// 2. Fallback handling
IF VO_Error THEN
    IF VI_Fallback_Mode = 1 THEN
        VO_Value := VI_Default_Value;
    END_IF;
    // If VI_Fallback_Mode = 0, VO_Value retains its last good value (L_Filtered)
    RETURN;
END_IF;

// 3. Calibration
L_Scaled := (L_Scaled * VI_Multiplier) + VI_Offset;

// 4. Moving Average Filter (ТЗ 1.2)
IF L_First_Scan THEN
    L_Filtered := L_Scaled;
    L_First_Scan := FALSE;
    L_Last_Time := VI_System_Time_MS;
    
    // Инициализация массива истории
    FOR L_i := 0 TO 9 DO
        L_History[L_i] := L_Scaled;
    END_FOR;
    L_History_Sum := L_Scaled * 10.0;
    L_History_Count := 10;
    L_History_Idx := 0;
END_IF;

L_DT := (SEL(VI_System_Time_MS >= L_Last_Time, VI_System_Time_MS - L_Last_Time, (4294967295 - L_Last_Time) + VI_System_Time_MS + 1));
IF VI_Filter_Time_MS = 0 THEN
    L_Filtered := L_Scaled;
    L_Last_Time := VI_System_Time_MS;
ELSIF L_DT >= (VI_Filter_Time_MS / 10) THEN // Обновляем 10 раз за время фильтрации
    // Вычитаем старое значение
    L_History_Sum := L_History_Sum - L_History[L_History_Idx];
    
    // Добавляем новое значение
    L_History[L_History_Idx] := L_Scaled;
    L_History_Sum := L_History_Sum + L_Scaled;
    
    // Сдвигаем индекс
    L_History_Idx := (L_History_Idx + 1) MOD 10;
    
    // Вычисляем среднее
    L_Filtered := L_History_Sum / 10.0;
    
    L_Last_Time := VI_System_Time_MS;
END_IF;

VO_Value := L_Filtered;
          
END_FUNCTION_BLOCK

FUNCTION_BLOCK FB_Sensor_Calibration
  VAR_INPUT
    VI_Sensor_ID : UDINT;
    VI_Reference_Value : REAL;
    VI_Current_Value : REAL;
    VI_Apply : BOOL;
  END_VAR
  VAR_OUTPUT
    VO_Offset : REAL;
    VO_Multiplier : REAL := 1.0;
    VO_Done : BOOL;
  END_VAR
  VAR
    L_Applied : BOOL;
  END_VAR

            IF VI_Apply AND NOT L_Applied THEN
    // Простая калибровка смещением (одноточечная)
    VO_Offset := VI_Reference_Value - VI_Current_Value;
    VO_Done := TRUE;
    L_Applied := TRUE;
ELSIF NOT VI_Apply THEN
    VO_Done := FALSE;
    L_Applied := FALSE;
END_IF;
          
END_FUNCTION_BLOCK

FUNCTION_BLOCK FB_Sensor_Calibration_Processor
  VAR_INPUT
    VI_Raw_Value : REAL;
    VI_Record : ST_Sensor_Calibration_Record;
  END_VAR
  VAR_OUTPUT
    VO_Calibrated_Value : REAL;
  END_VAR

            VO_Calibrated_Value := (VI_Raw_Value * VI_Record.multiplier) + VI_Record.offset;
          
END_FUNCTION_BLOCK

FUNCTION_BLOCK FB_Sensor_Distribution
  VAR_INPUT
    VI_Raw_Temp : REAL;
    VI_Raw_Hum : REAL;
    VI_Raw_CO2 : REAL;
  END_VAR
  VAR_OUTPUT
    VO_Temp_Heating : REAL;
    VO_Temp_Vent : REAL;
    VO_Hum_Vent : REAL;
    VO_CO2_Vent : REAL;
  END_VAR

            // Распределение данных по подсистемам
VO_Temp_Heating := VI_Raw_Temp;
VO_Temp_Vent    := VI_Raw_Temp;
VO_Hum_Vent     := VI_Raw_Hum;
VO_CO2_Vent     := VI_Raw_CO2;
          
END_FUNCTION_BLOCK

FUNCTION_BLOCK FB_Simulation_Manager
  VAR_INPUT
    VI_System_Time_MS : UDINT;
    VI_IsActivePLC : BOOL;
    VI_Scenario : E_SCENARIO_TYPE;
    VI_Config : ST_Scenario_Config;
  END_VAR
  VAR_OUTPUT
    VO_Sim_Lights : ARRAY[1..32] OF BOOL;
    VO_Sim_Active : BOOL;
    VO_Sim_Water_Leak : ARRAY[1..GVL_CONSTANTS.C_MAX_FLOOD_SENSORS] OF BOOL;
    VO_Sim_Gas_Leak : ARRAY[1..GVL_CONSTANTS.C_MAX_METHANE_SENSORS] OF REAL;
  END_VAR
  VAR
    L_Random : FB_Random_Generator;
    L_Last_Toggle : UDINT;
    L_i : INT;
    L_Rand_Val : UDINT;
    L_Test_Mode : BOOL := FALSE;
  END_VAR

            IF VI_Scenario = E_SCENARIO_TYPE.SCENARIO_AWAY AND VI_Config.Presence_Simulation_Enabled THEN
    VO_Sim_Active := TRUE;
    
    // Переключаем свет каждые 30 минут
    IF (VI_System_Time_MS - L_Last_Toggle) >= (GVL_CONSTANTS.C_MS_IN_MINUTE * 30) THEN
        L_Last_Toggle := VI_System_Time_MS;
        
        FOR L_i := 1 TO 32 DO
            L_Rand_Val := 1;
            VO_Sim_Lights[L_i] := (L_Rand_Val > 80); // 20% шанс включения
        END_FOR;
    END_IF;
ELSE
    VO_Sim_Active := FALSE;
    FOR L_i := 1 TO 32 DO VO_Sim_Lights[L_i] := FALSE; END_FOR;
END_IF;

// Симуляция аварий в тестовом режиме
IF L_Test_Mode THEN
    // Генерация случайных протечек (очень редко)
    L_Rand_Val := 1;
    IF L_Rand_Val = 42 THEN
        VO_Sim_Water_Leak[1] := TRUE;
    END_IF;
    
    // Симуляция утечки газа
    L_Rand_Val := 1;
    IF L_Rand_Val = 77 THEN
        VO_Sim_Gas_Leak[1] := 15.0; // 15% LEL
    END_IF;
ELSE
    FOR L_i := 1 TO GVL_CONSTANTS.C_MAX_FLOOD_SENSORS DO VO_Sim_Water_Leak[L_i] := FALSE; END_FOR;
    FOR L_i := 1 TO GVL_CONSTANTS.C_MAX_METHANE_SENSORS DO VO_Sim_Gas_Leak[L_i] := 0.0; END_FOR;
END_IF;
// >>> BULK_SYNC_ANCHOR: FB_Simulation_Manager <<<
          
END_FUNCTION_BLOCK

FUNCTION_BLOCK FB_Smoke_Detector
  VAR_INPUT
    VI_Smoke_Signal : BOOL;
  END_VAR
  VAR_OUTPUT
    VO_Smoke_Detected : BOOL;
  END_VAR

            VO_Smoke_Detected := VI_Smoke_Signal;
          
END_FUNCTION_BLOCK

FUNCTION_BLOCK FB_Socket_Manager
  VAR_INPUT
    VI_System_Time_MS : UDINT;
    VI_IsActivePLC : BOOL;
    VI_Scenario : E_SCENARIO_TYPE;
    VI_Fire_Alarm : BOOL;
    VI_Flood_Alarm : BOOL;
    VI_Security_Armed : BOOL;
  END_VAR
  VAR_OUTPUT
    VO_Socket_States : ARRAY[1..GVL_CONSTANTS.C_MAX_SOCKETS] OF BOOL;
    VO_Internal_States : ARRAY[1..GVL_CONSTANTS.C_MAX_SOCKETS] OF BOOL;
  END_VAR
  VAR_IN_OUT
    VI_Manual_Override : ARRAY[1..GVL_CONSTANTS.C_MAX_SOCKETS] OF BOOL;
    VI_Physical_Switches : ARRAY[1..GVL_CONSTANTS.C_MAX_SOCKETS] OF BOOL;
    VI_Rule_Actions : ARRAY[1..GVL_CONSTANTS.C_MAX_RULES] OF ST_Rule_Action;
    VI_IO_Modules_Online : ARRAY[1..GVL_CONSTANTS.C_MAX_MODULES] OF BOOL;
  END_VAR
  VAR
    fbSocketV2Staging : FB_Socket_V2_Staging;
    L_Socket_V2_Command_Shadow : ST_Socket_Command_V2;
    L_Socket_V2_State_Shadow : ST_Socket_State_V2;
    L_Socket_V2_Shadow_Diff_Found : BOOL;
    L_Socket_V2_Switch_Enabled : BOOL;
    L_Socket_V2_Path_Ready : BOOL;
    L_Socket_Using_Legacy_Fallback : BOOL;
    L_i : INT;
    L_j : INT;
    L_Rule_State : BOOL;
    L_Rule_Active : BOOL;
    L_Internal_State : ARRAY[1..GVL_CONSTANTS.C_MAX_SOCKETS] OF BOOL;
    L_Manual_Trig : ARRAY[1..GVL_CONSTANTS.C_MAX_SOCKETS] OF R_TRIG;
  END_VAR

            // Менеджер управления розетками.
// Обеспечивает работу по сценариям, правилам и аварийное отключение (без локальных выключателей розеток).


IF NOT VI_IsActivePLC THEN RETURN; END_IF;

L_Socket_V2_Shadow_Diff_Found := FALSE;
L_Socket_V2_Switch_Enabled := TRUE;
L_Socket_V2_Path_Ready := FALSE;
L_Socket_Using_Legacy_Fallback := TRUE;

// Проверка связи с модулями ввода-вывода
FOR L_i := 1 TO GVL_CONSTANTS.C_MAX_MODULES DO
    IF NOT VI_IO_Modules_Online[L_i] THEN
        // Переход в безопасное состояние при потере связи (отключение всех розеток)
        FOR L_j := 1 TO GVL_CONSTANTS.C_MAX_SOCKETS DO
            VO_Socket_States[L_j] := FALSE;
        END_FOR;
        RETURN;
    END_IF;
END_FOR;

FOR L_i := 1 TO GVL_CONSTANTS.C_MAX_SOCKETS DO
    L_Rule_Active := FALSE;
    L_Rule_State := FALSE;
    
    L_Manual_Trig[L_i](CLK := VI_Manual_Override[L_i]);
    
    // Ручное переключение
    IF L_Manual_Trig[L_i].Q THEN
        L_Internal_State[L_i] := NOT L_Internal_State[L_i];
    END_IF;

    // Проверка правил для текущей розетки
    FOR L_j := 1 TO GVL_CONSTANTS.C_MAX_RULES DO
        IF VI_Rule_Actions[L_j].Active AND VI_Rule_Actions[L_j].Target_ID = L_i THEN
            IF VI_Rule_Actions[L_j].Action_Type = E_Rule_Action_Type.ACTION_SET_SOCKET THEN
                L_Rule_Active := TRUE;
                L_Rule_State := (VI_Rule_Actions[L_j].Value > 0.5);
                L_Internal_State[L_i] := L_Rule_State; // Синхронизация внутреннего состояния
            ELSIF VI_Rule_Actions[L_j].Action_Type = E_Rule_Action_Type.ACTION_TOGGLE_SOCKET AND VI_Rule_Actions[L_j].Triggered THEN
                L_Internal_State[L_i] := NOT L_Internal_State[L_i]; // Toggle
            END_IF;
        END_IF;
    END_FOR;

    // Аварийное отключение
    IF VI_Fire_Alarm OR VI_Flood_Alarm THEN
        // Розетки 1-4 неотключаемые (холодильник, сервер и т.д.)
        IF L_i > 4 THEN
            VO_Socket_States[L_i] := FALSE;
        ELSE
            // Критические розетки сохраняют свое текущее внутреннее состояние, а не форсируются в TRUE
            VO_Socket_States[L_i] := L_Internal_State[L_i];
        END_IF;
    ELSIF VI_Scenario = E_SCENARIO_TYPE.SCENARIO_AWAY OR VI_Security_Armed THEN
        // Master Off
        IF L_i > 4 THEN
            VO_Socket_States[L_i] := FALSE;
        ELSE
            // Неотключаемые розетки могут управляться вручную
            VO_Socket_States[L_i] := L_Internal_State[L_i];
        END_IF;
    ELSE
        // Нормальный режим: состояние определяется внутренним состоянием (ручным или правилом)
        IF L_Rule_Active THEN
            VO_Socket_States[L_i] := L_Rule_State;
        ELSE
            VO_Socket_States[L_i] := L_Internal_State[L_i];
        END_IF;
    END_IF;
END_FOR;

VO_Internal_States := L_Internal_State;

// ========================================
// Socket V2 shadow execution (phase2)
// ========================================
fbSocketV2Staging(
    VI_Socket_ID := 1,
    VI_Enable := TRUE,
    VI_Target_State := VO_Socket_States[1],
    VI_Manual_Override := VI_Manual_Override[1],
    VI_Safety_Lock := (VI_Fire_Alarm OR VI_Flood_Alarm),
    VI_Scenario_ID := TO_INT(VI_Scenario),

    VI_Is_On := VO_Socket_States[1],
    VI_Manual_Override_Active := VI_Manual_Override[1],
    VI_Safety_Blocked := (VI_Fire_Alarm OR VI_Flood_Alarm),
    VI_Alarm_Active := (VI_Fire_Alarm OR VI_Flood_Alarm),

    VO_Command_Shadow => L_Socket_V2_Command_Shadow,
    VO_State_Shadow => L_Socket_V2_State_Shadow
);

// ========================================
// Socket V2 shadow validation
// ========================================
IF VO_Socket_States[1] <> L_Socket_V2_Command_Shadow.Target_State THEN
    L_Socket_V2_Shadow_Diff_Found := TRUE;
END_IF;
IF VO_Socket_States[1] <> L_Socket_V2_State_Shadow.Is_On THEN
    L_Socket_V2_Shadow_Diff_Found := TRUE;
END_IF;
IF (VI_Fire_Alarm OR VI_Flood_Alarm) <> L_Socket_V2_State_Shadow.Safety_Blocked THEN
    L_Socket_V2_Shadow_Diff_Found := TRUE;
END_IF;

// Guarded Socket V2 enable
IF L_Socket_V2_Switch_Enabled THEN
    IF NOT L_Socket_V2_Shadow_Diff_Found THEN
        L_Socket_V2_Path_Ready := TRUE;
        L_Socket_Using_Legacy_Fallback := FALSE;
    ELSE
        L_Socket_V2_Path_Ready := FALSE;
        L_Socket_Using_Legacy_Fallback := TRUE;
    END_IF;
ELSE
    L_Socket_V2_Path_Ready := FALSE;
    L_Socket_Using_Legacy_Fallback := TRUE;
END_IF;

// >>> BULK_SYNC_ANCHOR: FB_Socket_Manager <<<
          
END_FUNCTION_BLOCK

FUNCTION_BLOCK FB_Socket_V2_Staging
  VAR_INPUT
    VI_Socket_ID : INT;
    VI_Enable : BOOL;
    VI_Target_State : BOOL;
    VI_Manual_Override : BOOL;
    VI_Safety_Lock : BOOL;
    VI_Scenario_ID : INT;
    VI_Is_On : BOOL;
    VI_Manual_Override_Active : BOOL;
    VI_Safety_Blocked : BOOL;
    VI_Alarm_Active : BOOL;
  END_VAR
  VAR_OUTPUT
    VO_Command_Shadow : ST_Socket_Command_V2;
    VO_State_Shadow : ST_Socket_State_V2;
  END_VAR

            VO_Command_Shadow.Target_State := VI_Target_State;
VO_State_Shadow.Is_On := VI_Is_On;
VO_State_Shadow.Safety_Blocked := VI_Safety_Blocked;
          
END_FUNCTION_BLOCK

FUNCTION_BLOCK FB_State_Manager
  VAR_INPUT
    VI_System_Severity : E_System_Severity;
    VI_Root_Cause : E_System_Root_Cause;
    VI_Freeze_Risk : BOOL := FALSE;
  END_VAR
  VAR_OUTPUT
    VO_System_OK : BOOL;
    VO_System_Warning : BOOL;
    VO_System_Critical : BOOL;
    VO_Status_Msg : STRING(200);
    VO_System_Mode : E_System_Operating_Mode;
  END_VAR

            VO_System_OK := FALSE;
VO_System_Warning := FALSE;
VO_System_Critical := FALSE;
VO_Status_Msg := '';
VO_System_Mode := E_System_Operating_Mode.MODE_NORMAL;

CASE VI_System_Severity OF
    E_System_Severity.SEV_NORMAL:
        VO_System_OK := TRUE;
        VO_Status_Msg := 'Система в норме';
        VO_System_Mode := E_System_Operating_Mode.MODE_NORMAL;

    E_System_Severity.SEV_WARNING:
        VO_System_Warning := TRUE;
        VO_System_Mode := E_System_Operating_Mode.MODE_DEGRADED;
        CASE VI_Root_Cause OF
            E_System_Root_Cause.ROOT_WATER_LEAK:
                VO_Status_Msg := 'Предупреждение: протечка воды';
            E_System_Root_Cause.ROOT_CO_WARNING:
                VO_Status_Msg := 'Предупреждение: повышенный CO';
            ELSE
                VO_Status_Msg := 'Предупреждение системы';
        END_CASE;

    E_System_Severity.SEV_DEGRADED:
        VO_System_Warning := TRUE;
        VO_System_Mode := E_System_Operating_Mode.MODE_DEGRADED;
        CASE VI_Root_Cause OF
            E_System_Root_Cause.ROOT_SENSOR_FAULT:
                VO_Status_Msg := 'Деградация: ошибка датчика';
            E_System_Root_Cause.ROOT_IO_OFFLINE:
                VO_Status_Msg := 'Деградация: модуль IO недоступен';
            E_System_Root_Cause.ROOT_COMM_FAULT:
                VO_Status_Msg := 'Деградация: ошибка связи';
            E_System_Root_Cause.ROOT_WATCHDOG_FAULT:
                VO_Status_Msg := 'Деградация: watchdog fault';
            E_System_Root_Cause.ROOT_SUBSYSTEM_FAULT:
                VO_Status_Msg := 'Деградация: ошибка подсистемы';
            ELSE
                VO_Status_Msg := 'Деградация системы';
        END_CASE;

    E_System_Severity.SEV_CRITICAL:
        VO_System_Critical := TRUE;

        IF (VI_Root_Cause = E_System_Root_Cause.ROOT_GAS_LEAK OR
            VI_Root_Cause = E_System_Root_Cause.ROOT_CO_CRITICAL) AND
            VI_Freeze_Risk THEN
            VO_System_Mode := E_System_Operating_Mode.MODE_FREEZE_PROTECTION;
        ELSE
            VO_System_Mode := E_System_Operating_Mode.MODE_SAFE_STOP;
        END_IF;

        CASE VI_Root_Cause OF
            E_System_Root_Cause.ROOT_FIRE:
                VO_Status_Msg := 'АВАРИЯ: ПОЖАР';
            E_System_Root_Cause.ROOT_GAS_LEAK:
                VO_Status_Msg := 'АВАРИЯ: УТЕЧКА ГАЗА';
            E_System_Root_Cause.ROOT_CO_CRITICAL:
                VO_Status_Msg := 'АВАРИЯ: КРИТИЧЕСКИЙ CO';
            E_System_Root_Cause.ROOT_WATCHDOG_FAULT:
                VO_Status_Msg := 'АВАРИЯ: WATCHDOG';
            ELSE
                VO_Status_Msg := 'АВАРИЯ СИСТЕМЫ';
        END_CASE;
END_CASE;
// >>> BULK_SYNC_ANCHOR: FB_State_Manager <<<
          
END_FUNCTION_BLOCK

FUNCTION_BLOCK FB_State_Manager_MVP
  VAR_INPUT
    VI_Gas_Alarm : BOOL;
    VI_Fire_Alarm : BOOL;
    VI_Flood_Alarm : BOOL;
    VI_IO_Healthy : BOOL;
    VI_Freeze_Risk : BOOL;
    VI_Reset_Request : BOOL;
  END_VAR
  VAR_OUTPUT
    VO_System_Mode : INT;
  END_VAR
  VAR
    L_Fire_Latched : BOOL;
    L_Gas_Latched : BOOL;
    L_Flood_Latched : BOOL;
  END_VAR

            FUNCTION_BLOCK FB_State_Manager


// Fire latch
IF VI_Fire_Alarm THEN
    L_Fire_Latched := TRUE;
END_IF;
IF VI_Reset_Request AND NOT VI_Fire_Alarm THEN
    L_Fire_Latched := FALSE;
END_IF;

// Gas latch
IF VI_Gas_Alarm THEN
    L_Gas_Latched := TRUE;
END_IF;
IF VI_Reset_Request AND NOT VI_Gas_Alarm THEN
    L_Gas_Latched := FALSE;
END_IF;

// Flood latch
IF VI_Flood_Alarm THEN
    L_Flood_Latched := TRUE;
END_IF;
IF VI_Reset_Request AND NOT VI_Flood_Alarm THEN
    L_Flood_Latched := FALSE;
END_IF;

// Mode logic
IF L_Fire_Latched THEN
    VO_System_Mode := 2; // SAFE_STOP
ELSIF L_Flood_Latched THEN
    VO_System_Mode := 2;
ELSIF L_Gas_Latched THEN
    IF VI_Freeze_Risk THEN
        VO_System_Mode := 3; // FREEZE
    ELSE
        VO_System_Mode := 1; // DEGRADED
    END_IF;
ELSIF NOT VI_IO_Healthy THEN
    VO_System_Mode := 1;
ELSE
    VO_System_Mode := 0; // NORMAL
END_IF;
          
END_FUNCTION_BLOCK

FUNCTION_BLOCK FB_State_Replication
  VAR_INPUT
    VI_Local_Role : E_PLC_ROLE;
    VI_Sync_Req : BOOL;
    VI_Local_State : ST_System_State_Snapshot;
    VI_Remote_State : ST_System_State_Snapshot;
    VI_System_Time_MS : UDINT;
  END_VAR
  VAR_OUTPUT
    VO_State_Updated : BOOL;
    VO_Synced_State : ST_System_State_Snapshot;
  END_VAR
  VAR
    L_Sync_In_Progress : BOOL;
    L_Last_Sync_Time : UDINT;
    L_Periodic_Sync_Req : BOOL;
    L_Elapsed_Time : UDINT;
  END_VAR

            // Периодическая синхронизация (каждые 5 секунд)
L_Elapsed_Time := (SEL(VI_System_Time_MS >= L_Last_Sync_Time, VI_System_Time_MS - L_Last_Sync_Time, (4294967295 - L_Last_Sync_Time) + VI_System_Time_MS + 1));

IF L_Elapsed_Time > 5000 THEN
    L_Periodic_Sync_Req := TRUE;
    L_Last_Sync_Time := VI_System_Time_MS;
ELSE
    L_Periodic_Sync_Req := FALSE;
END_IF;

// State Replication Logic
// Синхронизация состояния между ПЛК (ТЗ 8.2)
IF (VI_Sync_Req OR L_Periodic_Sync_Req) AND NOT L_Sync_In_Progress THEN
    L_Sync_In_Progress := TRUE;
    
    // Разрешение конфликтов на основе версии состояния
    IF VI_Remote_State.Version > VI_Local_State.Version THEN
        VO_Synced_State := VI_Remote_State;
        VO_State_Updated := TRUE;
    ELSIF VI_Remote_State.Version = VI_Local_State.Version THEN
        // Если версии равны, приоритет у ведущего ПЛК
        IF VI_Local_Role = E_PLC_ROLE.ROLE_STANDBY THEN
            VO_Synced_State := VI_Remote_State;
            VO_State_Updated := TRUE;
        ELSE
            VO_Synced_State := VI_Local_State;
            VO_State_Updated := FALSE;
        END_IF;
    ELSE
        VO_Synced_State := VI_Local_State;
        VO_State_Updated := FALSE;
    END_IF;
ELSIF NOT (VI_Sync_Req OR L_Periodic_Sync_Req) THEN
    L_Sync_In_Progress := FALSE;
    VO_State_Updated := FALSE;
    VO_Synced_State := VI_Local_State;
END_IF;
          
END_FUNCTION_BLOCK

FUNCTION_BLOCK FB_State_Snapshot_Manager
  VAR_INPUT
    VI_System_Time_MS : UDINT;
    VI_Trigger_Event : BOOL;
    VI_Event_Code : WORD;
    VI_Current_State : ST_State_Snapshot;
  END_VAR
  VAR_OUTPUT
    VO_Snapshot_Saved : BOOL;
  END_VAR
  VAR
    L_Snapshot_Buffer : ARRAY[1..GVL_CONSTANTS.C_MAX_STATE_SNAPSHOTS] OF ST_State_Snapshot;
    L_Write_Idx : INT := 1;
  END_VAR

            IF VI_Trigger_Event THEN
    L_Snapshot_Buffer[L_Write_Idx] := VI_Current_State;
    L_Snapshot_Buffer[L_Write_Idx].timestamp_ms := VI_System_Time_MS;
    L_Snapshot_Buffer[L_Write_Idx].trigger_event_code := VI_Event_Code;
    
    L_Write_Idx := (L_Write_Idx MOD GVL_CONSTANTS.C_MAX_STATE_SNAPSHOTS) + 1;
    VO_Snapshot_Saved := TRUE;
ELSE
    VO_Snapshot_Saved := FALSE;
END_IF;
          
END_FUNCTION_BLOCK

FUNCTION_BLOCK FB_State_Snapshot_NVRAM
  VAR_INPUT
    VI_System_Time_MS : UDINT;
    VI_Save_Req : BOOL;
    VI_Snapshot : ST_State_Snapshot;
  END_VAR
  VAR_OUTPUT
    VO_Saved : BOOL;
    VO_Error : BOOL;
  END_VAR
  VAR
    L_FileName : STRING := '/home/root/snapshot.bin';
    L_State : INT := 0;
    fbFileOpen : FILE.Open;
    fbFileWrite : FILE.Write;
    fbFileClose : FILE.Close;
    L_FileHandle : FILE.HANDLE;
  END_VAR

            CASE L_State OF
    0: // Ожидание
        VO_Saved := FALSE;
        VO_Error := FALSE;
        IF VI_Save_Req THEN
            L_State := 10;
            fbFileOpen(xExecute := FALSE);
            fbFileWrite(xExecute := FALSE);
            fbFileClose(xExecute := FALSE);
        END_IF;
        
    10: // Открытие файла
        fbFileOpen(
            xExecute := TRUE,
            sFileName := L_FileName,
            eFileMode := FILE.MODE.MWRITE
        );
        IF fbFileOpen.xDone THEN
            L_FileHandle := fbFileOpen.hFile;
            fbFileOpen(xExecute := FALSE);
            L_State := 20;
        ELSIF fbFileOpen.xError THEN
            VO_Error := TRUE;
            L_State := 0;
        END_IF;
        
    20: // Запись
        fbFileWrite(
            xExecute := TRUE,
            hFile := L_FileHandle,
            pBuffer := ADR(VI_Snapshot),
            szSize := SIZEOF(VI_Snapshot)
        );
        IF fbFileWrite.xDone THEN
            fbFileWrite(xExecute := FALSE);
            L_State := 30;
        ELSIF fbFileWrite.xError THEN
            VO_Error := TRUE;
            L_State := 30; // Все равно закрываем файл
        END_IF;
        
    30: // Закрытие
        fbFileClose(
            xExecute := TRUE,
            hFile := L_FileHandle
        );
        IF fbFileClose.xDone THEN
            fbFileClose(xExecute := FALSE);
            IF NOT VO_Error THEN
                VO_Saved := TRUE;
            END_IF;
            L_State := 0;
        ELSIF fbFileClose.xError THEN
            VO_Error := TRUE;
            L_State := 0;
        END_IF;
END_CASE;
          
END_FUNCTION_BLOCK

FUNCTION_BLOCK FB_Supply_Ventilation_Controller
  VAR_INPUT
    VI_Outdoor_Temp : REAL;
    VI_Supply_Temp : REAL;
    VI_Target_Temp : REAL;
    VI_Config : ST_Ventilation_Unit_Config;
  END_VAR
  VAR_OUTPUT
    VO_Heater_Power : REAL;
    VO_Fan_Speed : BYTE;
  END_VAR
  VAR
    L_PID : FB_PID_Controller;
  END_VAR

            // ПИД-регулятор калорифера
L_PID(
    VI_SetPoint := VI_Target_Temp,
    VI_ProcessValue := VI_Supply_Temp, // Используем датчик притока
    VI_Kp := 5.0, VI_Tn := 60.0, VI_Tv := 0.0,
    VI_Y_Min := 0.0, VI_Y_Max := 100.0, VI_Cycle_Time_S := 1.0,
    VO_Output => VO_Heater_Power
);

VO_Fan_Speed := 50; // Базовая скорость
          
END_FUNCTION_BLOCK

FUNCTION_BLOCK FB_System_Health
  VAR_INPUT
    VI_Smoke_Detected : BOOL;
    VI_Gas_Detected : BOOL;
    VI_CO_Warning_Level : BOOL;
    VI_CO_Alarm_Level : BOOL;
    VI_Leak_Detected : BOOL;
    VI_Sensor_Fault : BOOL := FALSE;
    VI_IO_Offline : BOOL := FALSE;
    VI_Comm_Fault : BOOL := FALSE;
    VI_Watchdog_Fault : BOOL := FALSE;
    VI_Subsystem_Fault : BOOL := FALSE;
  END_VAR
  VAR_OUTPUT
    VO_System_Severity : E_System_Severity;
    VO_Root_Cause : E_System_Root_Cause;
    VO_Sensor_Fault : BOOL;
    VO_IO_Fault : BOOL;
    VO_Comm_Fault : BOOL;
    VO_Subsystem_Degraded : BOOL;
    VO_First_Fault_Active : BOOL;
    VO_First_Fault_Type : INT;
    VO_First_Fault_Source : INT;
  END_VAR

            VO_Sensor_Fault := VI_Sensor_Fault;
VO_IO_Fault := VI_IO_Offline;
VO_Comm_Fault := VI_Comm_Fault;
VO_Subsystem_Degraded := VI_Subsystem_Fault;

VO_System_Severity := E_System_Severity.SEV_NORMAL;
VO_Root_Cause := E_System_Root_Cause.ROOT_NONE;
VO_First_Fault_Active := FALSE;
VO_First_Fault_Type := 0;
VO_First_Fault_Source := 0;

// Priority: FIRE > GAS > CO > WATER > diagnostics
IF VI_Smoke_Detected THEN
    VO_System_Severity := E_System_Severity.SEV_CRITICAL;
    VO_Root_Cause := E_System_Root_Cause.ROOT_FIRE;
    VO_First_Fault_Active := TRUE;
    VO_First_Fault_Type := 5;

ELSIF VI_Gas_Detected THEN
    VO_System_Severity := E_System_Severity.SEV_CRITICAL;
    VO_Root_Cause := E_System_Root_Cause.ROOT_GAS_LEAK;
    VO_First_Fault_Active := TRUE;
    VO_First_Fault_Type := 6;

ELSIF VI_CO_Alarm_Level THEN
    VO_System_Severity := E_System_Severity.SEV_CRITICAL;
    VO_Root_Cause := E_System_Root_Cause.ROOT_CO_CRITICAL;
    VO_First_Fault_Active := TRUE;
    VO_First_Fault_Type := 7;

ELSIF VI_CO_Warning_Level THEN
    VO_System_Severity := E_System_Severity.SEV_WARNING;
    VO_Root_Cause := E_System_Root_Cause.ROOT_CO_WARNING;
    VO_First_Fault_Active := TRUE;
    VO_First_Fault_Type := 7;

ELSIF VI_Leak_Detected THEN
    VO_System_Severity := E_System_Severity.SEV_WARNING;
    VO_Root_Cause := E_System_Root_Cause.ROOT_WATER_LEAK;
    VO_First_Fault_Active := TRUE;
    VO_First_Fault_Type := 8;

ELSIF VI_Watchdog_Fault THEN
    VO_System_Severity := E_System_Severity.SEV_CRITICAL;
    VO_Root_Cause := E_System_Root_Cause.ROOT_WATCHDOG_FAULT;
    VO_First_Fault_Active := TRUE;
    VO_First_Fault_Type := 9;

ELSIF VI_IO_Offline THEN
    VO_System_Severity := E_System_Severity.SEV_DEGRADED;
    VO_Root_Cause := E_System_Root_Cause.ROOT_IO_OFFLINE;
    VO_First_Fault_Active := TRUE;
    VO_First_Fault_Type := 1;

ELSIF VI_Comm_Fault THEN
    VO_System_Severity := E_System_Severity.SEV_DEGRADED;
    VO_Root_Cause := E_System_Root_Cause.ROOT_COMM_FAULT;
    VO_First_Fault_Active := TRUE;
    VO_First_Fault_Type := 3;

ELSIF VI_Sensor_Fault THEN
    VO_System_Severity := E_System_Severity.SEV_DEGRADED;
    VO_Root_Cause := E_System_Root_Cause.ROOT_SENSOR_FAULT;
    VO_First_Fault_Active := TRUE;
    VO_First_Fault_Type := 2;

ELSIF VI_Subsystem_Fault THEN
    VO_System_Severity := E_System_Severity.SEV_DEGRADED;
    VO_Root_Cause := E_System_Root_Cause.ROOT_SUBSYSTEM_FAULT;
    VO_First_Fault_Active := TRUE;
    VO_First_Fault_Type := 4;
END_IF;
// >>> BULK_SYNC_ANCHOR: FB_System_Health <<<
          
END_FUNCTION_BLOCK

FUNCTION_BLOCK FB_System_Timer
  VAR_INPUT
    IN : BOOL;
    PT : TIME;
    VI_System_Time_MS : UDINT;
  END_VAR
  VAR_OUTPUT
    Q : BOOL;
    ET : TIME;
  END_VAR
  VAR
    L_Start_Time : UDINT;
    L_Running : BOOL;
  END_VAR

            // ==============================================================================
// Блок таймера, привязанный к системному времени (System Timer)
// Назначение:
// - Замена стандартного TON для обеспечения точной выдержки времени,
//   независимой от времени цикла ПЛК, с использованием единого системного времени.
// ==============================================================================



IF IN THEN
    IF NOT L_Running THEN
        L_Start_Time := VI_System_Time_MS;
        L_Running := TRUE;
        ET := T#0s;
        Q := FALSE;
    ELSE
        // Обработка переполнения UDINT (примерно 49 дней)
        ET := TO_TIME((SEL(VI_System_Time_MS >= L_Start_Time, VI_System_Time_MS - L_Start_Time, (4294967295 - L_Start_Time) + VI_System_Time_MS + 1)));
        
        IF ET >= PT THEN
            Q := TRUE;
            ET := PT;
        ELSE
            Q := FALSE;
        END_IF;
    END_IF;
ELSE
    L_Running := FALSE;
    ET := T#0s;
    Q := FALSE;
END_IF;
// >>> BULK_SYNC_ANCHOR: FB_System_Timer <<<
          
END_FUNCTION_BLOCK

FUNCTION_BLOCK FB_System_Timer_TOF
  VAR_INPUT
    IN : BOOL;
    PT : TIME;
    VI_System_Time_MS : UDINT;
  END_VAR
  VAR_OUTPUT
    Q : BOOL;
    ET : TIME;
  END_VAR
  VAR
    L_Start_Time : UDINT;
    L_Running : BOOL;
    L_Prev_IN : BOOL;
  END_VAR

            // ==============================================================================
// Блок таймера задержки выключения (System Timer TOF)
// Назначение:
// - Замена стандартного TOF для обеспечения точной выдержки времени,
//   независимой от времени цикла ПЛК, с использованием единого системного времени.
// ==============================================================================



IF IN THEN
    Q := TRUE;
    ET := T#0s;
    L_Running := FALSE;
ELSE
    IF L_Prev_IN THEN
        L_Start_Time := VI_System_Time_MS;
        L_Running := TRUE;
        ET := T#0s;
    END_IF;
    
    IF L_Running THEN
        // Обработка переполнения UDINT (примерно 49 дней)
        ET := TO_TIME((SEL(VI_System_Time_MS >= L_Start_Time, VI_System_Time_MS - L_Start_Time, (4294967295 - L_Start_Time) + VI_System_Time_MS + 1)));
        
        IF ET >= PT THEN
            Q := FALSE;
            ET := PT;
            L_Running := FALSE;
        ELSE
            Q := TRUE;
        END_IF;
    END_IF;
END_IF;

L_Prev_IN := IN;
          
END_FUNCTION_BLOCK

FUNCTION_BLOCK FB_Trend_Analyzer
  VAR_INPUT
    VI_Count : INT;
  END_VAR
  VAR_OUTPUT
    VO_Average : REAL;
    VO_Max : REAL;
    VO_Min : REAL;
    VO_Trend_Up : BOOL;
    VO_Trend_Down : BOOL;
  END_VAR
  VAR_IN_OUT
    VI_Data : ARRAY[1..GVL_CONSTANTS.C_MAX_TREND_DATA_POINTS] OF REAL;
  END_VAR
  VAR
    L_i : INT;
    L_Sum : REAL;
  END_VAR

            IF VI_Count > 0 AND VI_Count <= GVL_CONSTANTS.C_MAX_TREND_DATA_POINTS THEN
    VO_Max := VI_Data[1];
    VO_Min := VI_Data[1];
    L_Sum := 0.0;
    
    FOR L_i := 1 TO VI_Count DO
        IF VI_Data[L_i] > VO_Max THEN VO_Max := VI_Data[L_i]; END_IF;
        IF VI_Data[L_i] < VO_Min THEN VO_Min := VI_Data[L_i]; END_IF;
        L_Sum := L_Sum + VI_Data[L_i];
    END_FOR;
    
    VO_Average := L_Sum / INT_TO_REAL(VI_Count);
    
    IF VI_Count >= 2 THEN
        VO_Trend_Up := (VI_Data[VI_Count] > VI_Data[1]);
        VO_Trend_Down := (VI_Data[VI_Count] < VI_Data[1]);
    END_IF;
END_IF;
          
END_FUNCTION_BLOCK

FUNCTION_BLOCK FB_Trend_Logger
  VAR_INPUT
    VI_System_Time_MS : UDINT;
    VI_Config : ST_Trend_Config;
    VI_Current_Value : REAL;
  END_VAR
  VAR_OUTPUT
    VO_Data : ST_Trend_Data;
  END_VAR
  VAR
    L_Last_Log_Time : UDINT;
    L_Last_Value : REAL;
    L_Deviation : REAL;
  END_VAR

            IF NOT VI_Config.enabled THEN RETURN; END_IF;

// Логирование по изменению (Deadband) или по времени (раз в час)
L_Deviation := ABS(VI_Current_Value - L_Last_Value);
IF (L_Deviation >= (L_Last_Value * VI_Config.deviation_threshold_percent / 100.0)) OR 
   ((SEL(VI_System_Time_MS >= L_Last_Log_Time, VI_System_Time_MS - L_Last_Log_Time, (4294967295 - L_Last_Log_Time) + VI_System_Time_MS + 1)) >= GVL_CONSTANTS.C_MS_IN_HOUR) THEN
    
    // Запись в массив
    VO_Data.write_index := (VO_Data.record_count MOD 100) + 1;
    VO_Data.values[VO_Data.write_index] := VI_Current_Value;
    VO_Data.timestamps[VO_Data.write_index] := VI_System_Time_MS;

    VO_Data.record_count := VO_Data.record_count + 1;
    VO_Data.sum_values := VO_Data.sum_values + VI_Current_Value;
    
    L_Last_Value := VI_Current_Value;
    L_Last_Log_Time := VI_System_Time_MS;
END_IF;
          
END_FUNCTION_BLOCK

FUNCTION_BLOCK FB_TwoFactor_Auth
  VAR_INPUT
    VI_System_Time_MS : UDINT;
    VI_Start_Auth : BOOL;
    VI_Method : E_TwoFactor_Method;
    VI_User_Code : STRING(6);
    VI_Reset_Success : BOOL;
  END_VAR
  VAR_OUTPUT
    VO_State : ST_TwoFactor_Auth_State;
    VO_Send_Code_Req : BOOL;
    VO_Code_To_Send : STRING(6);
  END_VAR
  VAR
    L_Generated_Code : STRING(6) := '';
    L_Start_Time : UDINT;
    R_Trig_Start : R_TRIG;
    L_Prev_User_Code : STRING(6);
    L_Lockout_Start_Time : UDINT;
    fbHMAC : FB_HMAC_SHA1;
    L_Elapsed_Time : UDINT;
    L_Time_Step : UDINT;
    L_Message : ARRAY[0..7] OF BYTE;
    L_Key : ARRAY[0..63] OF BYTE;
    L_Offset : INT;
    L_Truncated_Hash : UDINT;
    L_i : INT;
    L_Current_TOTP : STRING(6);
    L_Prev_TOTP : STRING(6);
    L_Code_Valid : BOOL;
  END_VAR

            R_Trig_Start(CLK := VI_Start_Auth);

IF VI_Reset_Success THEN
    VO_State.Is_Success := FALSE;
END_IF;

IF R_Trig_Start.Q AND NOT VO_State.is_pending AND NOT VO_State.Is_Locked THEN
    VO_State.is_pending := TRUE;
    VO_State.Auth_Method := VI_Method;
    L_Start_Time := VI_System_Time_MS;
    VO_State.Attempts_Left := 3;
    VO_State.Is_Success := FALSE;
    VO_State.Is_Locked := FALSE;
    L_Prev_User_Code := '';
    
    IF VI_Method <> E_TwoFactor_Method.TF_METHOD_TOTP THEN
        // Генерируем одноразовый код через HMAC (без упрощенного алгоритма "по времени")
        L_Time_Step := VI_System_Time_MS / 30000;
        L_Key[0] := 16#31; L_Key[1] := 16#32; L_Key[2] := 16#33; L_Key[3] := 16#34; // Секрет-шаблон, заменяется из конфигурации
        FOR L_i := 0 TO 7 DO L_Message[7 - L_i] := TO_BYTE(SHR(L_Time_Step + L_Start_Time, L_i * 8) AND 16#FF); END_FOR;
        fbHMAC(Key := L_Key, KeyLength := 4, Message := L_Message, MessageLength := 8);
        L_Offset := TO_INT(fbHMAC.Hash[19] AND 16#0F);
        L_Truncated_Hash := (SHL(TO_UDINT(fbHMAC.Hash[L_Offset] AND 16#7F), 24) OR SHL(TO_UDINT(fbHMAC.Hash[L_Offset+1] AND 16#FF), 16) OR SHL(TO_UDINT(fbHMAC.Hash[L_Offset+2] AND 16#FF), 8) OR TO_UDINT(fbHMAC.Hash[L_Offset+3] AND 16#FF));
        L_Generated_Code := UDINT_TO_STRING(L_Truncated_Hash MOD 1000000);
        WHILE LEN(L_Generated_Code) < 6 DO
            L_Generated_Code := CONCAT('0', L_Generated_Code);
        END_WHILE;
        
        VO_Code_To_Send := L_Generated_Code;
        VO_Send_Code_Req := TRUE;
    ELSE
        // Для TOTP код не отправляем
        VO_Code_To_Send := '';
        VO_Send_Code_Req := FALSE;
    END_IF;
ELSE
    VO_Send_Code_Req := FALSE;
END_IF;

IF VO_State.is_pending THEN
    L_Elapsed_Time := (SEL(VI_System_Time_MS >= L_Start_Time, VI_System_Time_MS - L_Start_Time, (4294967295 - L_Start_Time) + VI_System_Time_MS + 1));

    IF L_Elapsed_Time < (GVL_CONSTANTS.C_MS_IN_MINUTE * 5) THEN
        VO_State.Time_Left_S := TO_UINT(((GVL_CONSTANTS.C_MS_IN_MINUTE * 5) - L_Elapsed_Time) / 1000);
    ELSE
        VO_State.Time_Left_S := 0;
    END_IF;
    
    IF VI_User_Code <> '' AND VI_User_Code <> L_Prev_User_Code THEN
        L_Code_Valid := FALSE;
        
        IF VI_Method = E_TwoFactor_Method.TF_METHOD_TOTP THEN
            // Вычисляем TOTP для текущего шага времени (30 секунд)
            L_Time_Step := VI_System_Time_MS / 30000; 
            
            // Подготовка ключа (в реальном проекте берется из GVL_CONFIG)
            L_Key[0] := 16#31; L_Key[1] := 16#32; L_Key[2] := 16#33; L_Key[3] := 16#34; // '1234'
            
            // Проверка текущего шага
            FOR L_i := 0 TO 7 DO L_Message[7 - L_i] := TO_BYTE(SHR(L_Time_Step, L_i * 8) AND 16#FF); END_FOR;
            fbHMAC(Key := L_Key, KeyLength := 4, Message := L_Message, MessageLength := 8);
            L_Offset := TO_INT(fbHMAC.Hash[19] AND 16#0F);
            L_Truncated_Hash := (SHL(TO_UDINT(fbHMAC.Hash[L_Offset] AND 16#7F), 24) OR SHL(TO_UDINT(fbHMAC.Hash[L_Offset+1] AND 16#FF), 16) OR SHL(TO_UDINT(fbHMAC.Hash[L_Offset+2] AND 16#FF), 8) OR TO_UDINT(fbHMAC.Hash[L_Offset+3] AND 16#FF));
            L_Current_TOTP := UDINT_TO_STRING(L_Truncated_Hash MOD 1000000);
            WHILE LEN(L_Current_TOTP) < 6 DO L_Current_TOTP := CONCAT('0', L_Current_TOTP); END_WHILE;
            
            // Проверка предыдущего шага (для компенсации рассинхронизации)
            FOR L_i := 0 TO 7 DO L_Message[7 - L_i] := TO_BYTE(SHR(L_Time_Step - 1, L_i * 8) AND 16#FF); END_FOR;
            fbHMAC(Key := L_Key, KeyLength := 4, Message := L_Message, MessageLength := 8);
            L_Offset := TO_INT(fbHMAC.Hash[19] AND 16#0F);
            L_Truncated_Hash := (SHL(TO_UDINT(fbHMAC.Hash[L_Offset] AND 16#7F), 24) OR SHL(TO_UDINT(fbHMAC.Hash[L_Offset+1] AND 16#FF), 16) OR SHL(TO_UDINT(fbHMAC.Hash[L_Offset+2] AND 16#FF), 8) OR TO_UDINT(fbHMAC.Hash[L_Offset+3] AND 16#FF));
            L_Prev_TOTP := UDINT_TO_STRING(L_Truncated_Hash MOD 1000000);
            WHILE LEN(L_Prev_TOTP) < 6 DO L_Prev_TOTP := CONCAT('0', L_Prev_TOTP); END_WHILE;
            
            IF VI_User_Code = L_Current_TOTP OR VI_User_Code = L_Prev_TOTP THEN
                L_Code_Valid := TRUE;
            END_IF;
        ELSE
            IF VI_User_Code = L_Generated_Code THEN
                L_Code_Valid := TRUE;
            END_IF;
        END_IF;
        
        IF L_Code_Valid THEN
            VO_State.Is_Success := TRUE;
            VO_State.is_pending := FALSE;
        ELSE
            IF VO_State.Attempts_Left > 0 THEN
                VO_State.Attempts_Left := VO_State.Attempts_Left - 1;
            END_IF;
            
            IF VO_State.Attempts_Left = 0 THEN
                VO_State.Is_Locked := TRUE;
                VO_State.is_pending := FALSE;
                L_Lockout_Start_Time := VI_System_Time_MS; // Блокировка на 5 минут
            END_IF;
        END_IF;
    END_IF;
    L_Prev_User_Code := VI_User_Code;
    
    IF L_Elapsed_Time > (GVL_CONSTANTS.C_MS_IN_MINUTE * 5) THEN
        VO_State.is_pending := FALSE; // Таймаут
    END_IF;
END_IF;

IF VO_State.Is_Locked THEN
    IF (SEL(VI_System_Time_MS >= L_Lockout_Start_Time, VI_System_Time_MS - L_Lockout_Start_Time, (4294967295 - L_Lockout_Start_Time) + VI_System_Time_MS + 1)) >= (GVL_CONSTANTS.C_MS_IN_MINUTE * 5) THEN
        VO_State.Is_Locked := FALSE;
    END_IF;
END_IF;
          
END_FUNCTION_BLOCK

FUNCTION_BLOCK FB_Valve_Test
  VAR_INPUT
    VI_System_Time_MS : UDINT;
    VI_Start_Test : BOOL;
    VI_Valve_ID : BYTE;
  END_VAR
  VAR_OUTPUT
    VO_Test_Active : BOOL;
    VO_Result : E_Valve_Test_Result;
    VO_Valve_Cmd : BOOL;
  END_VAR
  VAR
    L_Start_Time : UDINT;
    L_State : INT;
  END_VAR

            CASE L_State OF
    0: // Ожидание
        IF VI_Start_Test THEN
            VO_Test_Active := TRUE;
            VO_Result := E_Valve_Test_Result.TEST_IN_PROGRESS;
            L_Start_Time := VI_System_Time_MS;
            VO_Valve_Cmd := TRUE; // Открыть
            L_State := 1;
        END_IF;
    1: // Тест
        IF (SEL(VI_System_Time_MS >= L_Start_Time, VI_System_Time_MS - L_Start_Time, (4294967295 - L_Start_Time) + VI_System_Time_MS + 1)) > 5000 THEN
            VO_Valve_Cmd := FALSE; // Закрыть
            VO_Result := E_Valve_Test_Result.TEST_PASSED; // Заглушка, нужен контроль концевиков
            VO_Test_Active := FALSE;
            L_State := 0;
        END_IF;
END_CASE;
          
END_FUNCTION_BLOCK

FUNCTION_BLOCK FB_Valve_Test_Manager
  VAR_INPUT
    VI_System_Time_MS : UDINT;
    VI_IsActivePLC : BOOL;
  END_VAR
  VAR_OUTPUT
    VO_Test_Active : BOOL;
    VO_Current_Valve : INT;
    VO_Valve_Cmd : ARRAY[1..GVL_CONSTANTS.C_MAX_MANIFOLDS] OF BOOL;
    VO_Test_Results : ARRAY[1..GVL_CONSTANTS.C_MAX_MANIFOLDS] OF BOOL;
    VO_Status_Msg : STRING(200);
  END_VAR
  VAR_IN_OUT
    VI_Valve_Currents : ARRAY[1..GVL_CONSTANTS.C_MAX_MANIFOLDS] OF REAL;
    VI_Valve_End_Switches : ARRAY[1..GVL_CONSTANTS.C_MAX_MANIFOLDS] OF BOOL;
    VI_Config : ARRAY[1..GVL_CONSTANTS.C_MAX_MANIFOLDS] OF ST_Valve_Test_Config;
  END_VAR
  VAR
    L_State : INT;
    L_Current_Valve : INT := 1;
    L_Test_Start_Time : UDINT;
    L_Last_Test_Time : ARRAY[1..GVL_CONSTANTS.C_MAX_MANIFOLDS] OF UDINT;
    L_i : INT;
    L_Need_Test : BOOL;
    L_Elapsed_Time : UDINT;
  END_VAR

            IF NOT VI_IsActivePLC THEN RETURN; END_IF;

CASE L_State OF
    0: // Ожидание
        VO_Test_Active := FALSE;
        L_Need_Test := FALSE;
        
        // Поиск клапана, которому нужен тест (раз в неделю)
        FOR L_i := 1 TO GVL_CONSTANTS.C_MAX_MANIFOLDS DO
            IF VI_Config[L_i].enabled AND ((VI_System_Time_MS - L_Last_Test_Time[L_i]) > (VI_Config[L_i].test_interval_days * 86400000)) THEN
                L_Current_Valve := L_i;
                L_Need_Test := TRUE;
                EXIT;
            END_IF;
        END_FOR;
        
        IF L_Need_Test THEN
            L_State := 1;
            L_Test_Start_Time := VI_System_Time_MS;
            VO_Test_Active := TRUE;
            VO_Current_Valve := L_Current_Valve;
            VO_Valve_Cmd[L_Current_Valve] := TRUE; // Открываем
            VO_Status_Msg := CONCAT('ТЕСТ КЛАПАНА ', INT_TO_STRING(L_Current_Valve));
            VO_Test_Results[L_Current_Valve] := TRUE; // Сброс результата
        END_IF;
        
    1: // Тестирование (ожидание открытия)
        L_Elapsed_Time := (VI_System_Time_MS - L_Test_Start_Time);
        
        IF VI_Valve_End_Switches[L_Current_Valve] THEN
            // Концевик сработал до истечения таймаута
            // Проверка тока
            IF ABS(VI_Valve_Currents[L_Current_Valve] - VI_Config[L_Current_Valve].Nominal_Current) > (VI_Config[L_Current_Valve].Nominal_Current * 0.2) THEN
                VO_Test_Results[L_Current_Valve] := FALSE; // Ошибка по току
            END_IF;
            
            GVL_Retain.G_Valve_Test_Results[L_Current_Valve] := VO_Test_Results[L_Current_Valve];
            
            VO_Valve_Cmd[L_Current_Valve] := FALSE; // Закрываем
            L_Test_Start_Time := VI_System_Time_MS; // Перезапускаем таймер для проверки закрытия
            L_State := 2;
        ELSIF L_Elapsed_Time > TO_UDINT(VI_Config[L_Current_Valve].nominal_close_time_sec * 1000.0) THEN
            // Таймаут открытия (заклинивание)
            VO_Test_Results[L_Current_Valve] := FALSE; 
            GVL_Retain.G_Valve_Test_Results[L_Current_Valve] := FALSE;
            VO_Status_Msg := CONCAT('ОШИБКА: ЗАКЛИНИВАНИЕ КЛАПАНА ', INT_TO_STRING(L_Current_Valve));
            
            VO_Valve_Cmd[L_Current_Valve] := FALSE; // Закрываем
            L_Test_Start_Time := VI_System_Time_MS; // Перезапускаем таймер
            L_State := 2;
        END_IF;
        
    2: // Ожидание закрытия
        L_Elapsed_Time := (VI_System_Time_MS - L_Test_Start_Time);
        
        IF NOT VI_Valve_End_Switches[L_Current_Valve] THEN
            // Концевик разомкнулся (клапан закрыт)
            L_Last_Test_Time[L_Current_Valve] := VI_System_Time_MS;
            L_State := 0;
            IF VO_Test_Results[L_Current_Valve] THEN
                VO_Status_Msg := 'ТЕСТ ЗАВЕРШЕН УСПЕШНО';
            END_IF;
        ELSIF L_Elapsed_Time > TO_UDINT(VI_Config[L_Current_Valve].nominal_close_time_sec * 1000.0) THEN
            // Таймаут закрытия (заклинивание)
            VO_Test_Results[L_Current_Valve] := FALSE; 
            GVL_Retain.G_Valve_Test_Results[L_Current_Valve] := FALSE;
            VO_Status_Msg := CONCAT('ОШИБКА: НЕ ЗАКРЫЛСЯ КЛАПАН ', INT_TO_STRING(L_Current_Valve));
            
            L_Last_Test_Time[L_Current_Valve] := VI_System_Time_MS;
            L_State := 0;
        END_IF;
END_CASE;
          
END_FUNCTION_BLOCK

FUNCTION_BLOCK FB_Ventilation_System_Manager
  VAR_INPUT
    VI_System_Time_MS : UDINT;
    VI_IsActivePLC : BOOL;
    VI_Outdoor_Temp : REAL;
    VI_Current_Scenario : E_SCENARIO_TYPE;
    VI_System_Mode : E_System_Operating_Mode;
    VI_Config : ST_Ventilation_Global_Config;
    VI_Fire_Alarm : BOOL;
    VI_Gas_Alarm : BOOL;
    VI_PV3_Boost_Req : BOOL;
    VI_Supply_100_Req : BOOL;
    VI_Exhaust_100_Req : BOOL;
    VI_Supply_80_Req : BOOL;
    VI_Vent_Stop : BOOL;
    VI_IO_Modules_Online : ARRAY[1..GVL_CONSTANTS.C_MAX_MODULES] OF BOOL;
  END_VAR
  VAR_OUTPUT
    VO_Supply_Fans : ARRAY[1..GVL_CONSTANTS.C_MAX_SUPPLY_FANS] OF BYTE;
    VO_Exhaust_Fans : ARRAY[1..GVL_CONSTANTS.C_MAX_EXHAUST_FANS] OF BYTE;
    VO_Heater_Power : ARRAY[1..GVL_CONSTANTS.C_MAX_BOILERS] OF REAL;
    VO_Status_Msg : STRING(200);
  END_VAR
  VAR_IN_OUT
    VI_Supply_Temps : ARRAY[1..GVL_CONSTANTS.C_MAX_SUPPLY_TEMPS] OF REAL;
    VI_Room_Temps : ARRAY[1..16] OF REAL;
    VI_Room_Humidities : ARRAY[1..16] OF REAL;
    VI_Room_CO2 : ARRAY[1..16] OF REAL;
    VI_Wet_Zone_Active : ARRAY[1..GVL_CONSTANTS.C_MAX_WET_ZONES] OF BOOL;
    VI_Rule_Actions : ARRAY[1..GVL_CONSTANTS.C_MAX_RULES] OF ST_Rule_Action;
  END_VAR
  VAR
    L_Policy_Normal : BOOL;
    L_Policy_Safe_Stop : BOOL;
    L_Policy_Degraded : BOOL;
    L_Policy_Freeze_Protection : BOOL;
    L_i : INT;
    L_j : INT;
    L_Max_CO2 : REAL;
    L_Max_Hum : REAL;
    L_Base_Speed : BYTE;
    L_Target_Temp : REAL;
    L_PID_Heaters : ARRAY[1..GVL_CONSTANTS.C_MAX_BOILERS] OF FB_PID_Controller;
    L_Wet_Zone_Timers : ARRAY[1..GVL_CONSTANTS.C_MAX_WET_ZONES] OF FB_System_Timer_TOF;
    fbVentilationV2Staging : FB_Ventilation_V2_Staging;
    L_Vent_Command_Shadow : ST_Ventilation_Command_V2;
    L_Vent_State_Shadow : ST_Ventilation_State_V2;
    L_Vent_V2_Shadow_Diff_Found : BOOL;
    L_Vent_V2_Switch_Enabled : BOOL;
    L_Vent_V2_Path_Ready : BOOL;
    L_Vent_Using_Legacy_Fallback : BOOL;
  END_VAR

            // ========================================
// Ventilation policy layer (phase3/v2)
// ========================================
GVL_STATE.G_Ventilation_IO_Fault := FALSE;
GVL_STATE.G_Ventilation_Subsystem_Degraded := FALSE;
L_Vent_V2_Shadow_Diff_Found := FALSE;
L_Vent_V2_Switch_Enabled := TRUE;
L_Vent_V2_Path_Ready := FALSE;
L_Vent_Using_Legacy_Fallback := TRUE;
L_Policy_Normal := (VI_System_Mode = E_System_Operating_Mode.MODE_NORMAL);
L_Policy_Safe_Stop := (VI_System_Mode = E_System_Operating_Mode.MODE_SAFE_STOP);
L_Policy_Degraded := (VI_System_Mode = E_System_Operating_Mode.MODE_DEGRADED);
L_Policy_Freeze_Protection := (VI_System_Mode = E_System_Operating_Mode.MODE_FREEZE_PROTECTION);

IF NOT VI_IsActivePLC THEN
    FOR L_i := 1 TO GVL_CONSTANTS.C_MAX_SUPPLY_FANS DO
        VO_Supply_Fans[L_i] := 0;
        IF L_i <= GVL_CONSTANTS.C_MAX_SUPPLY_TEMPS THEN
            VO_Heater_Power[L_i] := 0.0;
        END_IF;
    END_FOR;
    FOR L_i := 1 TO GVL_CONSTANTS.C_MAX_EXHAUST_FANS DO
        VO_Exhaust_Fans[L_i] := 0;
    END_FOR;
    VO_Status_Msg := 'ВЕНТИЛЯЦИЯ: РЕЗЕРВНЫЙ ПЛК';
    RETURN;
END_IF;

// Проверка связи с модулями ввода-вывода
FOR L_i := 1 TO GVL_CONSTANTS.C_MAX_MODULES DO
    IF NOT VI_IO_Modules_Online[L_i] THEN
        GVL_STATE.G_Ventilation_IO_Fault := TRUE;
        // Переход в безопасное состояние при потере связи (отключение вентиляции)
        FOR L_j := 1 TO GVL_CONSTANTS.C_MAX_SUPPLY_FANS DO
            VO_Supply_Fans[L_j] := 0;
        END_FOR;
        FOR L_j := 1 TO GVL_CONSTANTS.C_MAX_EXHAUST_FANS DO
            VO_Exhaust_Fans[L_j] := 0;
        END_FOR;
        FOR L_j := 1 TO GVL_CONSTANTS.C_MAX_BOILERS DO
            VO_Heater_Power[L_j] := 0.0;
        END_FOR;
        VO_Status_Msg := 'ОШИБКА: Потеря связи с модулями ввода-вывода';
        RETURN;
    END_IF;
END_FOR;

// =========================
// SYSTEM MODE OVERRIDE
// =========================
// VENT_POLICY_ROUTING_PHASE3_V2
IF L_Policy_Safe_Stop THEN
    FOR L_i := 1 TO GVL_CONSTANTS.C_MAX_SUPPLY_FANS DO
        VO_Supply_Fans[L_i] := 0;
    END_FOR;
    FOR L_i := 1 TO GVL_CONSTANTS.C_MAX_EXHAUST_FANS DO
        VO_Exhaust_Fans[L_i] := 0;
    END_FOR;
    FOR L_i := 1 TO GVL_CONSTANTS.C_MAX_BOILERS DO
        VO_Heater_Power[L_i] := 0.0;
    END_FOR;
    VO_Status_Msg := 'ВЕНТИЛЯЦИЯ: ОСТАНОВЛЕНА POLICY SAFE_STOP';
    RETURN;
END_IF;

IF L_Policy_Degraded THEN
    FOR L_i := 1 TO GVL_CONSTANTS.C_MAX_SUPPLY_FANS DO
        VO_Supply_Fans[L_i] := 0;
    END_FOR;
    FOR L_i := 1 TO GVL_CONSTANTS.C_MAX_BOILERS DO
        VO_Heater_Power[L_i] := 0.0;
    END_FOR;
    GVL_STATE.G_Ventilation_Subsystem_Degraded := TRUE;
    VO_Status_Msg := 'ВЕНТИЛЯЦИЯ: DEGRADED POLICY';
END_IF;

IF L_Policy_Freeze_Protection THEN
    FOR L_i := 1 TO GVL_CONSTANTS.C_MAX_SUPPLY_FANS DO
        VO_Supply_Fans[L_i] := 0;
    END_FOR;
    FOR L_i := 1 TO GVL_CONSTANTS.C_MAX_EXHAUST_FANS DO
        VO_Exhaust_Fans[L_i] := 0;
    END_FOR;
    FOR L_i := 1 TO GVL_CONSTANTS.C_MAX_BOILERS DO
        VO_Heater_Power[L_i] := 0.0;
    END_FOR;
    VO_Status_Msg := 'ВЕНТИЛЯЦИЯ: FREEZE_PROTECTION POLICY (stop)';
    RETURN;
END_IF;

// MODE_FREEZE_PROTECTION пока оставляем на текущей штатной логике

// 1. Определение базовой скорости и целевой температуры по сценарию (ТЗ 7.1)
CASE VI_Current_Scenario OF
    E_SCENARIO_TYPE.SCENARIO_AWAY:
        L_Base_Speed := VI_Config.Scenario_Modes[3].Base_Fan_Speed;
        L_Target_Temp := VI_Config.Scenario_Modes[3].Target_Temp;
    E_SCENARIO_TYPE.SCENARIO_SLEEP:
        L_Base_Speed := VI_Config.Scenario_Modes[2].Base_Fan_Speed;
        L_Target_Temp := VI_Config.Scenario_Modes[2].Target_Temp;
    ELSE // PRESENCE, MORNING, EVENING
        L_Base_Speed := VI_Config.Scenario_Modes[1].Base_Fan_Speed;
        L_Target_Temp := VI_Config.Scenario_Modes[1].Target_Temp;
END_CASE;

// 2. Логика управления приточными установками (П-1, П-2, П-3)
FOR L_i := 1 TO GVL_CONSTANTS.C_MAX_SUPPLY_FANS DO
    // ПИД-регулирование мощности электрического калорифера
    IF L_i <= GVL_CONSTANTS.C_MAX_SUPPLY_TEMPS THEN
        L_PID_Heaters[L_i](
            VI_SetPoint := L_Target_Temp,
            VI_ProcessValue := VI_Supply_Temps[L_i], // Используем датчик температуры после калорифера
            VI_Kp := 4.0, VI_Tn := 120.0, VI_Tv := 0.0,
            VI_Y_Min := 0.0, VI_Y_Max := 100.0, VI_Cycle_Time_S := 1.0,
            VO_Output => VO_Heater_Power[L_i]
        );
    END_IF;

    // Определение скорости приточного вентилятора
    VO_Supply_Fans[L_i] := L_Base_Speed;
    
    // Обработка действий от Rule Engine
    FOR L_j := 1 TO GVL_CONSTANTS.C_MAX_RULES DO
        IF VI_Rule_Actions[L_j].Active AND VI_Rule_Actions[L_j].Target_ID = L_i THEN
            IF VI_Rule_Actions[L_j].Action_Type = E_Rule_Action_Type.ACTION_SET_VENTILATION THEN
                VO_Supply_Fans[L_i] := REAL_TO_BYTE(VI_Rule_Actions[L_j].Value);
            END_IF;
        END_IF;
    END_FOR;
    
    // Requests are observed but must not bypass policy directly.
    IF VI_Supply_100_Req OR VI_Supply_80_Req OR VI_Fire_Alarm OR VI_Vent_Stop OR VI_Gas_Alarm OR VI_PV3_Boost_Req THEN
        GVL_STATE.G_Ventilation_Subsystem_Degraded := TRUE;
    END_IF;
END_FOR;

// 3. Логика управления вытяжными установками (В-1 .. В-5)
FOR L_i := 1 TO GVL_CONSTANTS.C_MAX_EXHAUST_FANS DO
    VO_Exhaust_Fans[L_i] := L_Base_Speed;
    
    // ТЗ 4.0: Логика вытяжки в санузлах
    FOR L_j := 1 TO GVL_CONSTANTS.C_MAX_WET_ZONES DO
        IF VI_Config.wet_zone_to_exhaust_map[L_j] = L_i THEN
            // Включение по свету, выключение с задержкой 5 минут (используем TOF)
            L_Wet_Zone_Timers[L_j](IN := VI_Wet_Zone_Active[L_j], PT := T#5m, VI_System_Time_MS := VI_System_Time_MS);
            IF VI_Wet_Zone_Active[L_j] THEN
                VO_Exhaust_Fans[L_i] := 80; // Повышенная скорость при присутствии
            ELSIF L_Wet_Zone_Timers[L_j].Q THEN
                VO_Exhaust_Fans[L_i] := 50; // Скорость выбега (пока таймер TOF активен)
            END_IF;
        END_IF;
    END_FOR;

    // Requests are observed but must not bypass policy directly.
    IF (L_i = VI_Config.pv3_exhaust_index AND VI_PV3_Boost_Req) OR VI_Exhaust_100_Req OR VI_Fire_Alarm OR VI_Vent_Stop OR VI_Gas_Alarm THEN
        GVL_STATE.G_Ventilation_Subsystem_Degraded := TRUE;
    END_IF;
END_FOR;








// ========================================
// VENT_FINAL_CLAMP
// ========================================
IF L_Policy_Degraded THEN
    FOR L_i := 1 TO GVL_CONSTANTS.C_MAX_EXHAUST_FANS DO
        VO_Exhaust_Fans[L_i] := MIN(VO_Exhaust_Fans[L_i], VI_Config.Degraded_Exhaust_Limit);
    END_FOR;
END_IF;

// Ventilation V2 shadow runtime integration (diagnostic only)
fbVentilationV2Staging(
    VI_Zone_ID := 1,
    VI_Enable := (NOT L_Policy_Safe_Stop) AND (NOT L_Policy_Freeze_Protection) AND (NOT GVL_STATE.G_Ventilation_IO_Fault),
    VI_Fan_Speed_Setpoint := BYTE_TO_REAL(VO_Supply_Fans[1]),
    VI_Damper_Position_Setpoint := 0.0,
    VI_Heat_Recovery_Enabled := L_Policy_Normal,
    VI_Is_Active := (VO_Supply_Fans[1] > 0) OR (VO_Exhaust_Fans[1] > 0),
    VI_Fan_Speed_Actual := BYTE_TO_REAL(VO_Supply_Fans[1]),
    VI_Supply_Temp := VI_Supply_Temps[1],
    VI_Extract_Temp := VI_Room_Temps[1],
    VI_Filter_Dirty := FALSE,
    VI_Alarm_Active := GVL_STATE.G_Ventilation_IO_Fault OR GVL_STATE.G_Ventilation_Subsystem_Degraded,
    VO_Command_Shadow => L_Vent_Command_Shadow,
    VO_State_Shadow => L_Vent_State_Shadow
);

// Ventilation V2 shadow validation
IF ABS(BYTE_TO_REAL(VO_Supply_Fans[1]) - L_Vent_Command_Shadow.Fan_Speed_Setpoint) > 0.1 THEN
    L_Vent_V2_Shadow_Diff_Found := TRUE;
END_IF;
IF ABS(VI_Supply_Temps[1] - L_Vent_State_Shadow.Supply_Temp) > 0.1 THEN
    L_Vent_V2_Shadow_Diff_Found := TRUE;
END_IF;

// Guarded Ventilation V2 enable
IF L_Vent_V2_Switch_Enabled THEN
    IF NOT L_Vent_V2_Shadow_Diff_Found THEN
        L_Vent_V2_Path_Ready := TRUE;
        L_Vent_Using_Legacy_Fallback := FALSE;
    ELSE
        L_Vent_V2_Path_Ready := FALSE;
        L_Vent_Using_Legacy_Fallback := TRUE;
    END_IF;
ELSE
    L_Vent_V2_Path_Ready := FALSE;
    L_Vent_Using_Legacy_Fallback := TRUE;
END_IF;

// 4. Формирование статусного сообщения
IF L_Policy_Safe_Stop THEN
    VO_Status_Msg := 'ВЕНТИЛЯЦИЯ: ОСТАНОВЛЕНА POLICY SAFE_STOP';
ELSIF L_Policy_Freeze_Protection THEN
    VO_Status_Msg := 'ВЕНТИЛЯЦИЯ: FREEZE_PROTECTION POLICY (stop)';
ELSIF L_Policy_Degraded THEN
    VO_Status_Msg := 'ВЕНТИЛЯЦИЯ: DEGRADED POLICY';
ELSE
    VO_Status_Msg := 'Вентиляция работает в штатном режиме';
END_IF;
// >>> BULK_SYNC_ANCHOR: FB_Ventilation_System_Manager <<<
          
END_FUNCTION_BLOCK

FUNCTION_BLOCK FB_Ventilation_V2_Staging
  VAR_INPUT
    VI_Zone_ID : INT;
    VI_Enable : BOOL;
    VI_Fan_Speed_Setpoint : REAL;
    VI_Damper_Position_Setpoint : REAL;
    VI_Heat_Recovery_Enabled : BOOL;
    VI_Is_Active : BOOL;
    VI_Fan_Speed_Actual : REAL;
    VI_Supply_Temp : REAL;
    VI_Extract_Temp : REAL;
    VI_Filter_Dirty : BOOL;
    VI_Alarm_Active : BOOL;
  END_VAR
  VAR_OUTPUT
    VO_Command_Shadow : ST_Ventilation_Command_V2;
    VO_State_Shadow : ST_Ventilation_State_V2;
  END_VAR

            VO_Command_Shadow.Fan_Speed_Setpoint := VI_Fan_Speed_Setpoint;
VO_State_Shadow.Supply_Temp := VI_Supply_Temp;
          
END_FUNCTION_BLOCK

FUNCTION_BLOCK FB_Watchdog
  VAR_INPUT
    VI_System_Time_MS : UDINT;
    VI_Timeout_MS : UDINT := 2000;
  END_VAR
  VAR_OUTPUT
    VO_Alive : BOOL;
    VO_Watchdog_Fault : BOOL;
    VO_Cycle_DT_MS : UDINT;
  END_VAR
  VAR
    L_Initialized : BOOL := FALSE;
    L_Last_Call_MS : UDINT := 0;
    L_DT_MS : UDINT := 0;
  END_VAR

            IF NOT L_Initialized THEN
    L_Initialized := TRUE;
    L_Last_Call_MS := VI_System_Time_MS;
    VO_Cycle_DT_MS := 0;
    VO_Watchdog_Fault := FALSE;
    VO_Alive := TRUE;
    RETURN;
END_IF;

// Measure real time gap between successive calls
L_DT_MS := (SEL(VI_System_Time_MS >= L_Last_Call_MS, VI_System_Time_MS - L_Last_Call_MS, (4294967295 - L_Last_Call_MS) + VI_System_Time_MS + 1));
VO_Cycle_DT_MS := L_DT_MS;

// Fault if the task/cycle resumed after an abnormal pause
VO_Watchdog_Fault := (L_DT_MS > VI_Timeout_MS);
VO_Alive := NOT VO_Watchdog_Fault;

// Store current timestamp for next cycle
L_Last_Call_MS := VI_System_Time_MS;
// >>> BULK_SYNC_ANCHOR: FB_Watchdog <<<
          
END_FUNCTION_BLOCK

FUNCTION_BLOCK FB_Water_Leakage_Manager
  VAR_INPUT
    VI_System_Time_MS : UDINT;
    VI_IsActivePLC : BOOL;
    VI_Config : ST_Flood_Global_Config;
  END_VAR
  VAR_OUTPUT
    VO_Close_Valve_35 : BOOL;
    VO_Close_Valve_36 : BOOL;
    VO_Status_Msg : STRING(200);
    VO_Leak_Detected : BOOL;
    VO_Leak_Warning_Level : BOOL;
  END_VAR
  VAR_IN_OUT
    VI_Sensors : ARRAY[1..GVL_CONSTANTS.C_MAX_FLOOD_SENSORS] OF BOOL;
  END_VAR
  VAR
    L_i : INT;
    L_Sensor_Timers : ARRAY[1..GVL_CONSTANTS.C_MAX_FLOOD_SENSORS] OF FB_System_Timer;
    L_Any_Leak : BOOL;
    L_Any_Warning : BOOL;
  END_VAR

            IF NOT VI_IsActivePLC THEN RETURN; END_IF;

L_Any_Leak := FALSE;
L_Any_Warning := FALSE;

FOR L_i := 1 TO GVL_CONSTANTS.C_MAX_FLOOD_SENSORS DO
    L_Sensor_Timers[L_i](
        IN := VI_Sensors[L_i],
        PT := TO_TIME(VI_Config.min_duration_ms + VI_Config.warning_duration_ms),
        VI_System_Time_MS := VI_System_Time_MS
    );

    IF L_Sensor_Timers[L_i].ET >= TO_TIME(VI_Config.min_duration_ms) THEN
        L_Any_Warning := TRUE;

        IF L_Sensor_Timers[L_i].Q THEN
            L_Any_Leak := TRUE;

            IF VI_Config.sensor_to_valve_map[L_i] = 1 THEN
                VO_Close_Valve_35 := TRUE;
            ELSIF VI_Config.sensor_to_valve_map[L_i] = 2 THEN
                VO_Close_Valve_36 := TRUE;
            END_IF;
        END_IF;
    END_IF;
END_FOR;

// Health signals
VO_Leak_Detected := L_Any_Leak;
VO_Leak_Warning_Level := L_Any_Warning;

// Status
IF L_Any_Leak THEN
    VO_Status_Msg := 'АВАРИЯ: ПРОТЕЧКА ВОДЫ. КЛАПАНЫ ЗАКРЫТЫ.';
ELSIF L_Any_Warning THEN
    VO_Status_Msg := 'ПРЕДУПРЕЖДЕНИЕ: ОБНАРУЖЕНА ВОДА.';
ELSE
    VO_Status_Msg := 'Система контроля протечек в норме';
    VO_Close_Valve_35 := FALSE;
    VO_Close_Valve_36 := FALSE;
END_IF;
// >>> BULK_SYNC_ANCHOR: FB_Water_Leakage_Manager <<<
          
END_FUNCTION_BLOCK

FUNCTION_BLOCK FB_Water_Valve_Controller
  VAR_INPUT
    VI_System_Time : UDINT;
    VI_IsActivePLC : BOOL;
    VI_Flood_Alarm : BOOL;
  END_VAR
  VAR_INPUT
    VI_Operator_ID : STRING(10);
    VI_Force : BOOL;
  END_VAR
  VAR_INPUT
    VI_Operator_ID : STRING(10);
    VI_Force : BOOL;
  END_VAR
  VAR_OUTPUT
    VO_Valve_Closed : BOOL;
    VO_Status_Msg : STRING(200);
  END_VAR

            IF VI_Flood_Alarm AND VI_IsActivePLC THEN
    VO_Valve_Closed := TRUE;
    VO_Status_Msg := 'КЛАПАН ЗАКРЫТ ПО ПРОТЕЧКЕ';
END_IF;

METHOD OpenValve : BOOL

IF VI_IsActivePLC OR VI_Force THEN
    VO_Valve_Closed := FALSE;
    OpenValve := TRUE;
END_IF;
END_METHOD

METHOD CloseValve : BOOL

VO_Valve_Closed := TRUE;
CloseValve := TRUE;
END_METHOD

METHOD GetStatus : BYTE
GetStatus := TO_BYTE(SEL(VO_Valve_Closed, 0, 1));
END_METHOD
          
END_FUNCTION_BLOCK

FUNCTION_BLOCK FB_Zone_Access_Manager
  VAR_INPUT
    VI_System_Time_MS : UDINT;
    VI_Operator_ID : STRING(10);
    VI_Target_Zone : INT;
    VI_Rights : ST_Operator_Zone_Rights;
  END_VAR
  VAR_OUTPUT
    VO_Access_Granted : BOOL;
  END_VAR

            // Проверка прав доступа к зоне
IF VI_Target_Zone >= 1 AND VI_Target_Zone <= 32 THEN
    // Если глобальный уровень доступа высокий (например, CONFIG или FULL), разрешаем доступ ко всем зонам
    IF VI_Rights.global_access_level >= TO_BYTE(E_Zone_Access_Level.ZONE_ACCESS_CONFIG) THEN
        VO_Access_Granted := TRUE;
    ELSE
        // Иначе проверяем битовую маску для конкретной зоны
        // Бит 0 соответствует зоне 1, бит 1 - зоне 2 и т.д.
        VO_Access_Granted := (VI_Rights.zone_masks AND SHL(DWORD#1, VI_Target_Zone - 1)) <> 0;
    END_IF;
ELSE
    VO_Access_Granted := FALSE;
END_IF;
          
END_FUNCTION_BLOCK

PROGRAM PRG_Heating
  VAR
    fbHeatingManager : FB_Heating_System_Manager;
    fbDHWManager : FB_DHW_Manager;
    L_i : INT;
    L_Zone_Valves_8 : ARRAY[1..8] OF BOOL;
    L_Boiler_Modulation_REAL : ARRAY[1..GVL_CONSTANTS.C_MAX_BOILERS] OF REAL;
  END_VAR

            FOR L_i := 1 TO GVL_CONSTANTS.C_MAX_BOILERS DO
    L_Boiler_Modulation_REAL[L_i] := TO_REAL(GVL_IO.AI_Boiler_Modulation[L_i]);
END_FOR;

// 9. Управление климатом (Отопление)
fbHeatingManager(
    VI_System_Time_MS := GVL_STATUS.G_System_Time_MS,
    VI_Current_TOD := GVL_STATUS.G_Current_TOD,
    VI_IsActivePLC := GVL_STATUS.G_Is_Active_PLC,
    VI_Outdoor_Temp := GVL_STATE.G_Outdoor_Temp,
    VI_Floor_Temps := GVL_STATE.G_Floor_Temps,
    VI_Room_Temps := GVL_STATE.G_Room_Temps,
    VI_Config := GVL_CONFIG.G_Heating_Config,
    VI_Zone_Configs := GVL_CONFIG.G_HMI_FloorHeating_Configs,
    VI_Tariff := GVL_CONFIG.G_HMI_Tariff_Settings,
    VI_Current_Hour := TO_UINT(GVL_STATUS.G_Time_Of_Day_MS / GVL_CONSTANTS.C_MS_IN_HOUR),
    VI_Manifold_Pressures := GVL_STATE.G_Manifold_Pressures,
    VI_Manifold_Currents := GVL_STATE.G_Manifold_Currents,
    VI_Manifold_Temps_Supply := GVL_STATE.G_Manifold_T_Supply,
    VI_Manifold_Temps_Return := GVL_STATE.G_Manifold_T_Return,
    VI_Boiler_Flame_Status := GVL_STATE.G_Boiler_Flame,
    VI_Boiler_Error_Status := GVL_STATE.G_Boiler_Error,
    VI_Boiler_OT_Online := GVL_STATE.G_Boiler_OT_Online,
    VI_Boiler_Modulation := L_Boiler_Modulation_REAL,
    VI_Rule_Actions := GVL_STATE.G_Rule_Actions,
    VI_Boiler_Stop := GVL_COMMAND.G_Boiler_Stop,
    VI_IO_Modules_Online := GVL_STATUS.G_IO_Modules_Online,
    VI_DHW_Heating_Demand := fbDHWManager.VO_Heating_Pump,
    VI_DHW_Target_Temp := GVL_CONFIG.G_DHW_Config.Target_Temp,
    VI_Current_Scenario := GVL_STATUS.G_Current_Scenario,
    VI_System_Mode := GVL_STATE.G_System_Mode,
    VI_Emergency_Stop := GVL_STATE.G_Safety_Emergency_Stop,
    VI_Gas_Safety_Stop := GVL_STATE.G_Safety_Gas_Latched,
    VI_Scenario_Configs := GVL_CONFIG.G_HMI_Scenario_Configs,
    VI_Manifold_End_Switches := GVL_STATE.G_Manifold_End_Switches,
    VI_Valve_Test_Config := GVL_CONFIG.G_Valve_Test_Config,
    VO_Manifold_Valves => GVL_STATE.G_Manifold_Valves,
    VO_Manifold_Pumps => GVL_STATE.G_Manifold_Pumps,
    VO_Zone_Valves => L_Zone_Valves_8,
    VO_Boiler_OT_Enable => GVL_STATE.G_Boiler_OT_Enable,
    VO_Boiler_OT_Setpoint => GVL_STATE.G_Boiler_OT_Setpoint,
    VO_Backup_Circulation_Pump => GVL_STATE.G_Backup_Circulation_Pump,
    VO_Electric_Heater_Enable => GVL_STATE.G_Electric_Heater_Enable,
    VO_Freeze_Risk_Status => GVL_STATE.G_Safety_Freeze_Risk,
    VO_Status => GVL_STATUS.G_Manifold_Status,
    VO_Boiler_Status => GVL_STATUS.G_Boiler_Status
);

// 12. Управление ГВС
fbDHWManager(
    VI_System_Time_MS := GVL_STATUS.G_System_Time_MS,
    VI_Current_TOD := GVL_STATUS.G_Current_TOD,
    VI_IsActivePLC := GVL_STATUS.G_Is_Active_PLC,
    VI_Temp := GVL_STATE.G_DHW_Temp,
    VI_Pressure := GVL_STATE.G_DHW_Pressure,
    VI_Config := GVL_CONFIG.G_DHW_Config,
    VI_Current_Day_Of_Week := GVL_STATUS.G_Current_Day,
    VI_IO_Modules_Online := GVL_STATUS.G_IO_Modules_Online,
    VI_Reset_Errors := GVL_COMMAND.G_Reset_Errors,
    VI_Emergency_Stop := GVL_STATE.G_Safety_Emergency_Stop,
    VO_Heating_Pump => GVL_STATE.G_DHW_Heating_Pump,
    VO_Circ_Pump => GVL_STATE.G_DHW_Circ_Pump,
    VO_Status => GVL_STATUS.G_DHW_Status
);

// Integrated freeze-hardware diagnostics and maintenance gating
GVL_STATUS.G_Diagnostics.Backup_Pump_Out_Of_Service := NOT GVL_CONFIG.G_Backup_Circulation_Pump_In_Service;
GVL_STATUS.G_Diagnostics.Electric_Heater_Out_Of_Service := NOT GVL_CONFIG.G_Electric_Heater_In_Service;
IF NOT GVL_CONFIG.G_Backup_Circulation_Pump_In_Service THEN
    GVL_STATE.G_Backup_Circulation_Pump := FALSE;
END_IF;
IF NOT GVL_CONFIG.G_Electric_Heater_In_Service THEN
    GVL_STATE.G_Electric_Heater_Enable := FALSE;
END_IF;

GVL_STATE.G_Freeze_Hardware_Degraded := GVL_STATUS.G_Diagnostics.Backup_Pump_Fault OR GVL_STATUS.G_Diagnostics.Electric_Heater_Fault;
GVL_STATE.G_Freeze_Hardware_Failed := GVL_STATUS.G_Diagnostics.Backup_Pump_Fault AND GVL_STATUS.G_Diagnostics.Electric_Heater_Fault;

IF GVL_STATE.G_Freeze_Hardware_Failed THEN
    GVL_STATE.G_Backup_Circulation_Pump := FALSE;
    GVL_STATE.G_Electric_Heater_Enable := FALSE;
    GVL_STATE.G_Safety_Freeze_Risk := TRUE;
END_IF;

FOR L_i := 1 TO GVL_CONSTANTS.C_MAX_MANIFOLDS DO
    GVL_STATUS.G_Diagnostics.Manifold_Pump_Out_Of_Service[L_i] := NOT GVL_CONFIG.G_Manifold_Pump_In_Service[L_i];
    IF NOT GVL_CONFIG.G_Manifold_Pump_In_Service[L_i] THEN
        GVL_STATE.G_Manifold_Pumps[L_i] := FALSE;
    END_IF;
END_FOR;
GVL_STATUS.G_Diagnostics.DHW_Heating_Pump_Out_Of_Service := NOT GVL_CONFIG.G_DHW_Heating_Pump_In_Service;
IF NOT GVL_CONFIG.G_DHW_Heating_Pump_In_Service THEN
    GVL_STATE.G_DHW_Heating_Pump := FALSE;
END_IF;
GVL_STATUS.G_Diagnostics.DHW_Circ_Pump_Out_Of_Service := NOT GVL_CONFIG.G_DHW_Circ_Pump_In_Service;
IF NOT GVL_CONFIG.G_DHW_Circ_Pump_In_Service THEN
    GVL_STATE.G_DHW_Circ_Pump := FALSE;
END_IF;
// >>> BULK_SYNC_ANCHOR: PRG_Heating <<<


// HEATING ADAPTER COPY OUT
FOR L_i := 1 TO 8 DO
    GVL_STATE.G_Zone_Valves[L_i] := L_Zone_Valves_8[L_i];
END_FOR;
          
END_PROGRAM

PROGRAM PRG_IO_Read
  VAR
    L_i : INT;
    L_Debounce_Time : TIME := T#100MS;
    fbDebounce_Switches : ARRAY[1..8] OF FB_System_Timer;
    fbDebounce_Motion : ARRAY[1..8] OF FB_System_Timer;
    fbDebounce_Security_Open : ARRAY[1..GVL_CONSTANTS.C_MAX_SECURITY_SENSORS] OF FB_System_Timer;
    fbDebounce_Security_Glass : ARRAY[1..GVL_CONSTANTS.C_MAX_SECURITY_SENSORS] OF FB_System_Timer;
    fbDebounce_Flood : ARRAY[1..GVL_CONSTANTS.C_MAX_FLOOD_SENSORS] OF FB_System_Timer;
    fbDebounce_Smoke : ARRAY[1..GVL_CONSTANTS.C_MAX_SMOKE_SENSORS] OF FB_System_Timer;
    fbDebounce_Group_2F : FB_System_Timer;
    fbIO_Watchdog_1 : FB_IO_Module_Watchdog;
    fbIO_Watchdog_2 : FB_IO_Module_Watchdog;
    L_IO_Error_Active : BOOL;
  END_VAR

            // 0. КОНТРОЛЬ СВЯЗИ С МОДУЛЯМИ ВВОДА-ВЫВОДА (Watchdog)
fbIO_Watchdog_1(
    VI_System_Time_MS := GVL_STATUS.G_System_Time_MS,
    VI_Module_ID := 1,
    VI_Heartbeat_Signal := GVL_IO.DI_Module_1_Heartbeat,
    VI_Timeout_MS := 2000
);

fbIO_Watchdog_2(
    VI_System_Time_MS := GVL_STATUS.G_System_Time_MS,
    VI_Module_ID := 2,
    VI_Heartbeat_Signal := GVL_IO.DI_Module_2_Heartbeat,
    VI_Timeout_MS := 2000
);

GVL_STATUS.G_IO_Modules_Online[1] := fbIO_Watchdog_1.VO_Module_Online;
GVL_STATUS.G_IO_Modules_Online[2] := fbIO_Watchdog_2.VO_Module_Online;

L_IO_Error_Active := fbIO_Watchdog_1.VO_Error_Active OR fbIO_Watchdog_2.VO_Error_Active;

IF L_IO_Error_Active THEN
    GVL_COMMAND.G_Gas_Valve_Close := TRUE;
    GVL_COMMAND.G_Close_Valve_35 := TRUE;
    GVL_COMMAND.G_Close_Valve_36 := TRUE;
    FOR L_i := 1 TO GVL_CONSTANTS.C_MAX_MANIFOLDS DO GVL_STATE.G_Manifold_Pumps[L_i] := FALSE; END_FOR;
END_IF;

// 1. ЧТЕНИЕ И ФИЛЬТРАЦИЯ ВХОДОВ
FOR L_i := 1 TO 8 DO
    fbDebounce_Switches[L_i](IN := GVL_IO.DI_Lighting_Switches[L_i], PT := L_Debounce_Time, VI_System_Time_MS := GVL_STATUS.G_System_Time_MS);
    GVL_STATE.G_Physical_Switches[L_i] := fbDebounce_Switches[L_i].Q;
    
    fbDebounce_Motion[L_i](IN := GVL_IO.DI_Motion_Sensors[L_i], PT := L_Debounce_Time, VI_System_Time_MS := GVL_STATUS.G_System_Time_MS);
    GVL_STATE.G_Motion_Sensors[L_i] := fbDebounce_Motion[L_i].Q;
END_FOR;

FOR L_i := 1 TO GVL_CONSTANTS.C_MAX_SOCKETS DO
    // В текущей концепции локальные физические выключатели розеток не используются.
    // Состояние оставляем FALSE для обратной совместимости структуры.
    GVL_STATE.G_Socket_Switches[L_i] := FALSE;
END_FOR;

FOR L_i := 1 TO GVL_CONSTANTS.C_MAX_SECURITY_SENSORS DO
    fbDebounce_Security_Open[L_i](IN := GVL_IO.DI_Security_Open[L_i], PT := L_Debounce_Time, VI_System_Time_MS := GVL_STATUS.G_System_Time_MS);
    fbDebounce_Security_Glass[L_i](IN := GVL_IO.DI_Security_Glass[L_i], PT := L_Debounce_Time, VI_System_Time_MS := GVL_STATUS.G_System_Time_MS);
END_FOR;
fbDebounce_Group_2F(IN := GVL_IO.DI_Security_2F_Group, PT := L_Debounce_Time, VI_System_Time_MS := GVL_STATUS.G_System_Time_MS);

FOR L_i := 1 TO GVL_CONSTANTS.C_MAX_DOOR_SENSORS DO
    IF GVL_CONFIG.G_Door_Map[L_i] > 0 AND GVL_CONFIG.G_Door_Map[L_i] <= GVL_CONSTANTS.C_MAX_SECURITY_SENSORS THEN
        GVL_STATE.G_Door_Sensors[L_i] := fbDebounce_Security_Open[GVL_CONFIG.G_Door_Map[L_i]].Q;
    END_IF;
END_FOR;

FOR L_i := 1 TO 8 DO
    IF GVL_CONFIG.G_Window_Map[L_i] > 0 THEN
        IF GVL_CONFIG.G_Window_Map[L_i] <= GVL_CONSTANTS.C_MAX_SECURITY_SENSORS THEN
            GVL_STATE.G_Window_Sensors[L_i] := fbDebounce_Security_Open[GVL_CONFIG.G_Window_Map[L_i]].Q;
        ELSIF GVL_CONFIG.G_Window_Map[L_i] <= (GVL_CONSTANTS.C_MAX_SECURITY_SENSORS * 2) THEN
            GVL_STATE.G_Window_Sensors[L_i] := fbDebounce_Security_Glass[GVL_CONFIG.G_Window_Map[L_i] - GVL_CONSTANTS.C_MAX_SECURITY_SENSORS].Q;
        END_IF;
    END_IF;
END_FOR;
GVL_STATE.G_Window_Sensors[16] := fbDebounce_Group_2F.Q;

FOR L_i := 1 TO GVL_CONSTANTS.C_MAX_FLOOD_SENSORS DO
    fbDebounce_Flood[L_i](IN := GVL_IO.DI_Flood_Sensors[L_i], PT := L_Debounce_Time, VI_System_Time_MS := GVL_STATUS.G_System_Time_MS);
    GVL_STATE.G_Water_Sensors[L_i] := fbDebounce_Flood[L_i].Q;
END_FOR;

FOR L_i := 1 TO GVL_CONSTANTS.C_MAX_SMOKE_SENSORS DO
    fbDebounce_Smoke[L_i](IN := GVL_IO.DI_Smoke_Sensors[L_i], PT := L_Debounce_Time, VI_System_Time_MS := GVL_STATUS.G_System_Time_MS);
    GVL_STATE.G_Smoke_Sensors[L_i] := fbDebounce_Smoke[L_i].Q;
END_FOR;

IF GVL_IO.AI_Temp_Outdoor.wStatus = 0 THEN
    GVL_STATE.G_Outdoor_Temp := GVL_IO.AI_Temp_Outdoor.rValue;
END_IF;

FOR L_i := 1 TO GVL_CONSTANTS.C_MAX_SUPPLY_TEMPS DO
    IF GVL_IO.AI_Supply_Temps[L_i].wStatus = 0 THEN
        GVL_STATE.G_Supply_Temps[L_i] := GVL_IO.AI_Supply_Temps[L_i].rValue;
    END_IF;
END_FOR;

FOR L_i := 1 TO 8 DO
    GVL_STATE.G_Room_Hum[L_i] := GVL_IO.AI_Room_Hum[L_i];
    GVL_STATE.G_Room_CO2[L_i] := GVL_IO.AI_Room_CO2[L_i];
END_FOR;
FOR L_i := 1 TO 8 DO
    IF GVL_CONFIG.G_FloorTemp_Map[L_i] > 0 AND GVL_CONFIG.G_FloorTemp_Map[L_i] <= 8 THEN
        GVL_STATE.G_Floor_Temps[L_i] := GVL_IO.AI_Floor_Temps[GVL_CONFIG.G_FloorTemp_Map[L_i]];
    END_IF;
    IF GVL_CONFIG.G_RoomTemp_Map[L_i] > 0 AND GVL_CONFIG.G_RoomTemp_Map[L_i] <= 8 THEN
        GVL_STATE.G_Room_Temps[L_i] := GVL_IO.AI_Room_Temps[GVL_CONFIG.G_RoomTemp_Map[L_i]];
    END_IF;
END_FOR;

FOR L_i := 1 TO GVL_CONSTANTS.C_MAX_MANIFOLDS DO
    GVL_STATE.G_Manifold_Pressures[L_i] := INT_TO_REAL(GVL_IO.AI_Manifold_Pressures[L_i]) / 10.0;
    GVL_STATE.G_Manifold_Currents[L_i] := INT_TO_REAL(GVL_IO.AI_Manifold_Currents[L_i]) / 100.0;
    IF GVL_IO.AI_Manifold_Temps_Supply[L_i].wStatus = 0 THEN
        GVL_STATE.G_Manifold_T_Supply[L_i] := GVL_IO.AI_Manifold_Temps_Supply[L_i].rValue;
    END_IF;
    GVL_STATE.G_Manifold_T_Return[L_i] := INT_TO_REAL(GVL_IO.AI_Manifold_Temps_Return[L_i]) / 10.0;
    GVL_STATE.G_Manifold_End_Switches[L_i] := GVL_IO.DI_Manifold_End_Switches[L_i];
END_FOR;

FOR L_i := 1 TO GVL_CONSTANTS.C_MAX_METHANE_SENSORS DO
    IF GVL_IO.AI_Methane_LEL[L_i].wStatus = 0 THEN
        GVL_STATE.G_Methane_Sensors[L_i] := GVL_IO.AI_Methane_LEL[L_i].rValue;
    END_IF;
END_FOR;
GVL_STATE.G_Boiler_Flame := GVL_IO.AI_Boiler_Flame_Status;
GVL_STATE.G_Boiler_Error := GVL_IO.DI_Boiler_Error;
// --- SAFETY bootstrap mapping (temporary, will be normalized later if dedicated managers exist) ---
GVL_STATE.G_Safety_Gas_Alarm := FALSE;
GVL_STATE.G_Safety_Leak_Alarm := FALSE;
GVL_STATE.G_Safety_Smoke_Alarm := FALSE;

// Временное безопасное поведение:
// до подключения реального драйвера/шлюза OpenTherm считаем канал котла недоступным.
FOR L_i := 1 TO GVL_CONSTANTS.C_MAX_BOILERS DO
    GVL_STATE.G_Boiler_OT_Online[L_i] := FALSE;
END_FOR;
GVL_STATE.G_CO_Sensors := GVL_IO.AI_CO_PPM;

GVL_STATE.G_DHW_Temp := GVL_IO.AI_DHW_Temp;
GVL_STATE.G_DHW_Pressure := GVL_IO.AI_DHW_Pressure;

// Water zonal valve feedback mapping
GVL_STATE.G_Water_Zone_Open_FB := GVL_IO.DI_Water_Zone_Open_FB;
GVL_STATE.G_Water_Zone_Close_FB := GVL_IO.DI_Water_Zone_Close_FB;

GVL_STATUS.G_Diagnostics.Backup_Pump_Fault := FALSE;
GVL_STATUS.G_Diagnostics.Electric_Heater_Fault := FALSE;
// >>> BULK_SYNC_ANCHOR: PRG_IO_Read <<<
          
END_PROGRAM

PROGRAM PRG_IO_Write
  VAR
    L_i : INT;
  END_VAR

            // 2. ЗАПИСЬ ВЫХОДОВ (GVL_STATE -> GVL_IO)

// 2.1. Отопление (Термоэлектрические приводы)
FOR L_i := 1 TO 8 DO
    GVL_IO.DO_Zone_Valves[L_i] := GVL_STATE.G_Zone_Valves[L_i];
END_FOR;

// 2.2. Коллекторы (Насосы и смесительные клапаны)
FOR L_i := 1 TO GVL_CONSTANTS.C_MAX_MANIFOLDS DO
    GVL_IO.DO_Manifold_Pumps[L_i] := GVL_STATE.G_Manifold_Pumps[L_i];
    // Масштабирование 0.0-1.0 в 0-1000 для аналогового выхода (0-10В)
    GVL_IO.AO_Manifold_Valves[L_i] := REAL_TO_UINT(GVL_STATE.G_Manifold_Valves[L_i] * 1000.0);
END_FOR;

// 2.4. Вентиляция
FOR L_i := 1 TO GVL_CONSTANTS.C_MAX_SUPPLY_FANS DO
    GVL_IO.AO_Supply_Fans[L_i] := REAL_TO_UINT(GVL_STATE.G_Supply_Fans[L_i] * 100.0);
END_FOR;
FOR L_i := 1 TO GVL_CONSTANTS.C_MAX_EXHAUST_FANS DO
    GVL_IO.AO_Exhaust_Fans[L_i] := REAL_TO_UINT(GVL_STATE.G_Exhaust_Fans[L_i] * 100.0);
END_FOR;

// 2.5. ГВС
GVL_IO.DO_DHW_Heating_Pump := GVL_STATE.G_DHW_Heating_Pump;
GVL_IO.DO_DHW_Circ_Pump := GVL_STATE.G_DHW_Circ_Pump;
IF GVL_STATUS.G_Is_Active_PLC THEN
    GVL_IO.DO_Backup_Circulation_Pump := GVL_STATE.G_Backup_Circulation_Pump;
    GVL_IO.DO_Electric_Heater_Enable := GVL_STATE.G_Electric_Heater_Enable;
ELSE
    GVL_IO.DO_Backup_Circulation_Pump := FALSE;
    GVL_IO.DO_Electric_Heater_Enable := FALSE;
END_IF;

// 2.6. Освещение и шторы (полноценная выдача в физические каналы 0-10В)
FOR L_i := 1 TO 8 DO
    GVL_IO.AO_Lighting_Levels[L_i] := BYTE_TO_UINT(GVL_STATE.G_Lighting_Levels[L_i]) * 10;
END_FOR;
FOR L_i := 1 TO GVL_CONSTANTS.C_MAX_BLINDS DO
    GVL_IO.AO_Blinds_Positions[L_i] := BYTE_TO_UINT(GVL_STATE.G_Blinds_Positions[L_i]) * 10;
END_FOR;

// 2.7. Аварийные выходы (Сирены и клапаны)
IF GVL_ALARM.G_Gas_Fire_Siren AND GVL_ALARM.G_Gas_Alarm_Active THEN
    GVL_IO.DO_Gas_Siren := TRUE;
ELSE
    GVL_IO.DO_Gas_Siren := FALSE;
END_IF;

IF GVL_ALARM.G_Gas_Fire_Siren AND GVL_ALARM.G_Fire_Alarm_Active THEN
    GVL_IO.DO_Fire_Siren := TRUE;
ELSE
    GVL_IO.DO_Fire_Siren := FALSE;
END_IF;

IF GVL_ALARM.G_Security_Siren THEN
    GVL_IO.DO_Security_Siren := TRUE;
ELSE
    GVL_IO.DO_Security_Siren := FALSE;
END_IF;

IF GVL_COMMAND.G_Close_Valve_35 THEN
    GVL_IO.DO_Water_Valve_35_Close := TRUE;
ELSE
    GVL_IO.DO_Water_Valve_35_Close := FALSE;
END_IF;

IF GVL_COMMAND.G_Close_Valve_36 THEN
    GVL_IO.DO_Water_Valve_36_Close := TRUE;
ELSE
    GVL_IO.DO_Water_Valve_36_Close := FALSE;
END_IF;

IF GVL_COMMAND.G_Gas_Valve_Close THEN
    GVL_IO.DO_Gas_Valve_Close := TRUE;
ELSE
    GVL_IO.DO_Gas_Valve_Close := FALSE;
END_IF;

// 2.8. Управление доступом (Периметральная автоматика)
GVL_IO.DO_Gate_Open := GVL_COMMAND.G_Gate_Open;
GVL_IO.DO_Wicket_Open := GVL_COMMAND.G_Wicket_Open;
GVL_IO.DO_Lock_1_Open := GVL_COMMAND.G_Lock_1_Open;
GVL_IO.DO_Lock_1_Close := GVL_COMMAND.G_Lock_1_Close;
GVL_IO.DO_Lock_2_Open := GVL_COMMAND.G_Lock_2_Open;
GVL_IO.DO_Lock_2_Close := GVL_COMMAND.G_Lock_2_Close;

// 2.9. Розетки
GVL_IO.DO_Sockets := GVL_STATE.G_Socket_States;

// Selective zonal water recovery outputs
FOR L_i := 1 TO 32 DO
    GVL_IO.DO_Water_Zone_Enable[L_i] := GVL_STATE.G_Water_Zone_Enable[L_i];
END_FOR;
// >>> BULK_SYNC_ANCHOR: PRG_IO_Write <<<
          
END_PROGRAM

PROGRAM PRG_Lighting
  VAR
    L_i : INT;
    fbLightingManager : FB_Lighting_Blinds_Manager;
    fbSocketManager : FB_Socket_Manager;
    L_Manual_Light_Override_32 : ARRAY[1..32] OF BYTE;
    L_Sim_Lights_32 : ARRAY[1..32] OF BOOL;
    L_Physical_Switches_32 : ARRAY[1..32] OF BOOL;
    L_Motion_Sensors_32 : ARRAY[1..32] OF BOOL;
  END_VAR

            FOR L_i := 1 TO 32 DO
    IF L_i <= 16 THEN
        L_Manual_Light_Override_32[L_i] := GVL_COMMAND.G_Lighting_Override[L_i];
        L_Sim_Lights_32[L_i] := GVL_STATE.G_Sim_Lights[L_i];
        L_Physical_Switches_32[L_i] := GVL_STATE.G_Physical_Switches[L_i];
        L_Motion_Sensors_32[L_i] := GVL_STATE.G_Motion_Sensors[L_i];
    ELSE
        L_Manual_Light_Override_32[L_i] := 0;
        L_Sim_Lights_32[L_i] := FALSE;
        L_Physical_Switches_32[L_i] := FALSE;
        L_Motion_Sensors_32[L_i] := FALSE;
    END_IF;
END_FOR;

// 10. Управление освещением и шторами
fbLightingManager(
    VI_System_Time_MS := GVL_STATUS.G_System_Time_MS,
    VI_IsActivePLC := GVL_STATUS.G_Is_Active_PLC,
    VI_Current_Scenario := GVL_STATUS.G_Current_Scenario,
    VI_Away_Level := 1,
    VI_Simulation_Active := GVL_STATUS.G_Sim_Active,
    VI_Manual_Light_Override := L_Manual_Light_Override_32,
    VI_Manual_Blinds_Override := GVL_COMMAND.G_Blinds_Override,
    VI_Simulation_Lights := L_Sim_Lights_32,
    VI_Physical_Switches := L_Physical_Switches_32,
    VI_Motion_Sensors := L_Motion_Sensors_32,
    VI_Is_Night := GVL_STATUS.G_Is_Night,
    VI_Rule_Actions := GVL_STATE.G_Rule_Actions,
    VI_IO_Modules_Online := GVL_STATUS.G_IO_Modules_Online,
    VI_Wet_Zone_Map := GVL_CONFIG.G_Wet_Zone_Map,
    VI_Scenario_Configs := GVL_CONFIG.G_HMI_Scenario_Configs,
    VO_Lighting_Levels => GVL_STATE.G_Lighting_Levels,
    VO_Blinds_Positions => GVL_STATE.G_Blinds_Positions
);

// 11.5 Управление розетками
fbSocketManager(
    VI_System_Time_MS := GVL_STATUS.G_System_Time_MS,
    VI_IsActivePLC := GVL_STATUS.G_Is_Active_PLC,
    VI_Scenario := GVL_STATUS.G_Current_Scenario,
    VI_Manual_Override := GVL_COMMAND.G_Socket_Override,
    VI_Physical_Switches := GVL_STATE.G_Socket_Switches,
    VI_Rule_Actions := GVL_STATE.G_Rule_Actions,
    VI_Fire_Alarm := GVL_ALARM.G_Fire_Alarm_Active,
    VI_Flood_Alarm := GVL_ALARM.G_Flood_Alarm_Active,
    VI_Security_Armed := GVL_ALARM.G_Security_Armed,
    VI_IO_Modules_Online := GVL_STATUS.G_IO_Modules_Online,
    VO_Socket_States => GVL_STATE.G_Socket_States
);

// Evacuation lighting override
IF GVL_STATE.G_Evacuation_Lighting_Active THEN
    FOR L_i := 1 TO 8 DO
        IF (L_i MOD 2) = 0 THEN
            GVL_STATE.G_Lighting_Levels[L_i] := 100;
        ELSE
            GVL_STATE.G_Lighting_Levels[L_i] := 0;
        END_IF;
    END_FOR;
END_IF;


// Directional evacuation override
IF GVL_STATE.G_Evacuation_Lighting_Active THEN
    FOR L_i := 1 TO GVL_CONFIG.C_MAX_LIGHT_ZONES DO
        CASE GVL_STATE.G_Evac_Guidance[L_i] OF
            -1: // опасная зона — гасим или минимизируем
                GVL_STATE.G_Lighting_Levels[L_i] := 0;
            1: // направление к выходу — держим включенным
                GVL_STATE.G_Lighting_Levels[L_i] := 100;
        ELSE
            // нейтрально — мягкое мигание
            GVL_STATE.G_Lighting_Levels[L_i] := SEL((L_i MOD 2) = 0, 0, 100);
        END_CASE;
    END_FOR;
END_IF;
// >>> BULK_SYNC_ANCHOR: PRG_Lighting <<<
          
END_PROGRAM

PROGRAM PRG_PLC_A

            // Вызов основной программы
PRG_System();
// >>> BULK_SYNC_ANCHOR: PRG_PLC_A <<<
          
END_PROGRAM

PROGRAM PRG_PLC_B

            // Вызов основной программы
PRG_System();
// >>> BULK_SYNC_ANCHOR: PRG_PLC_B <<<
          
END_PROGRAM

PROGRAM PRG_Safety
  VAR
    fbWaterLeakageManager : FB_Water_Leakage_Manager;
    fbGasSmokeManager : FB_Gas_Smoke_Manager;
    L_i : INT;
    L_Water_Test_Active : BOOL;
    L_Water_Test_Deadline : UDINT;
    L_Gas_Test_Active : BOOL;
    L_Gas_Test_Deadline : UDINT;
    L_Water_Valve_Last_Exercise_MS : ARRAY[1..32] OF UDINT;
    L_Water_Valve_Exercise_Until_MS : ARRAY[1..32] OF UDINT;
    L_Water_Zone_Close_Last_Retry_MS : ARRAY[1..32] OF UDINT;
  END_VAR

            // 7.5 Система защиты от протечек
fbWaterLeakageManager(
    VI_System_Time_MS := GVL_STATUS.G_System_Time_MS,
    VI_IsActivePLC := GVL_STATUS.G_Is_Active_PLC,
    VI_Sensors := GVL_STATE.G_Water_Sensors,
    VI_Config := GVL_CONFIG.G_HMI_Flood_Config,
    VO_Close_Valve_35 => GVL_COMMAND.G_Close_Valve_35,
    VO_Close_Valve_36 => GVL_COMMAND.G_Close_Valve_36,
    VO_Status_Msg => GVL_STATUS.G_Flood_Status_Msg,
    VO_Leak_Detected => GVL_HEALTH_BRIDGE.G_Leak_Detected,
    VO_Leak_Warning_Level => GVL_HEALTH_BRIDGE.G_Leak_Warning_Level
);
GVL_ALARM.G_Flood_Alarm_Active := GVL_HEALTH_BRIDGE.G_Leak_Detected;

// 8. Пожарная и газовая безопасность (Приоритет 1)
fbGasSmokeManager(
    VI_System_Time_MS := GVL_STATUS.G_System_Time_MS,
    VI_IsActivePLC := GVL_STATUS.G_Is_Active_PLC,
    VI_Methane_LEL := GVL_STATE.G_Methane_Sensors,
    VI_CO_PPM := GVL_STATE.G_CO_Sensors,
    VI_Smoke_Sensors := GVL_STATE.G_Smoke_Sensors,
    VI_Mute_Request := GVL_CONFIG.G_HMI_Mute_Alarm,
    VO_Smoke_Detected => GVL_HEALTH_BRIDGE.G_Smoke_Detected,
    VO_Gas_Detected => GVL_HEALTH_BRIDGE.G_Gas_Detected,
    VO_CO_Warning_Level => GVL_HEALTH_BRIDGE.G_CO_Warning_Level,
    VO_CO_Alarm_Level => GVL_HEALTH_BRIDGE.G_CO_Alarm_Level,
    VO_Siren_Active => GVL_ALARM.G_Gas_Fire_Siren,
    VO_Status_Msg => GVL_STATUS.G_Gas_Status_Msg,
    VO_Gas_Valve_Close => GVL_COMMAND.G_Gas_Valve_Close,
    VO_Boiler_Stop => GVL_COMMAND.G_Boiler_Stop,
    VO_Supply_100_Req => GVL_COMMAND.G_Supply_100_Req,
    VO_Supply_80_Req => GVL_COMMAND.G_Supply_80_Req,
    VO_Vent_PV3_Boost => GVL_COMMAND.G_Vent_PV3_Boost,
    VO_Exhaust_100_Req => GVL_COMMAND.G_Exhaust_100_Req,
    VO_Vent_Stop => GVL_COMMAND.G_Vent_Stop
);
GVL_ALARM.G_Fire_Alarm_Active := GVL_HEALTH_BRIDGE.G_Smoke_Detected;
GVL_ALARM.G_Gas_Alarm_Active := GVL_HEALTH_BRIDGE.G_Gas_Detected OR GVL_HEALTH_BRIDGE.G_CO_Alarm_Level;
// Нормализация приоритетов и защёлкнутых safety-команд
// 1. Пожар/дым имеет приоритет над газовой вентиляцией
IF GVL_STATE.G_Safety_Smoke_Latched THEN
    GVL_COMMAND.G_Boiler_Stop := TRUE;
    GVL_COMMAND.G_Vent_Stop := TRUE;
    GVL_COMMAND.G_Supply_100_Req := FALSE;
    GVL_COMMAND.G_Supply_80_Req := FALSE;
    GVL_COMMAND.G_Vent_PV3_Boost := FALSE;
    GVL_COMMAND.G_Exhaust_100_Req := FALSE;

    // Эвакуация: разблокируем электронные замки для свободного выхода людей.
    GVL_COMMAND.G_Lock_1_Open := TRUE;
    GVL_COMMAND.G_Lock_1_Close := FALSE;
    GVL_COMMAND.G_Lock_2_Open := TRUE;
    GVL_COMMAND.G_Lock_2_Close := FALSE;
END_IF;

// 2. Газовая авария защёлкивает закрытие газа и стоп котлов
IF GVL_STATE.G_Safety_Gas_Latched THEN
    GVL_COMMAND.G_Gas_Valve_Close := TRUE;
    GVL_COMMAND.G_Boiler_Stop := TRUE;
END_IF;

// 3. Протечка защёлкивает перекрытие воды
IF GVL_STATE.G_Safety_Leak_Latched THEN
    GVL_COMMAND.G_Close_Valve_35 := TRUE;
    GVL_COMMAND.G_Close_Valve_36 := TRUE;
END_IF;

// Формирование зон опасности для направленной эвакуации через программную конфигурацию.
// Монтаж может быть выполнен произвольно: фактический вход ПЛК не определяет зону напрямую.
FOR L_i := 1 TO GVL_CONFIG.C_MAX_LIGHT_ZONES DO
    GVL_STATE.G_Evac_Hazard_Zone[L_i] := FALSE;
END_FOR;

FOR L_i := 1 TO GVL_CONSTANTS.C_MAX_SMOKE_SENSORS DO
    IF GVL_STATE.G_Smoke_Sensors[L_i] THEN
        IF (GVL_CONFIG.G_Evac_Smoke_Zone_Map[L_i] >= 1) AND (GVL_CONFIG.G_Evac_Smoke_Zone_Map[L_i] <= GVL_CONFIG.C_MAX_LIGHT_ZONES) THEN
            GVL_STATE.G_Evac_Hazard_Zone[GVL_CONFIG.G_Evac_Smoke_Zone_Map[L_i]] := TRUE;
        END_IF;
    END_IF;
END_FOR;

FOR L_i := 1 TO GVL_CONSTANTS.C_MAX_FLOOD_SENSORS DO
    IF GVL_STATE.G_Water_Sensors[L_i] THEN
        IF (GVL_CONFIG.G_Evac_Leak_Zone_Map[L_i] >= 1) AND (GVL_CONFIG.G_Evac_Leak_Zone_Map[L_i] <= GVL_CONFIG.C_MAX_LIGHT_ZONES) THEN
            GVL_STATE.G_Evac_Hazard_Zone[GVL_CONFIG.G_Evac_Leak_Zone_Map[L_i]] := TRUE;
        END_IF;
    END_IF;
END_FOR;

FOR L_i := 1 TO GVL_CONSTANTS.C_MAX_METHANE_SENSORS DO
    IF GVL_STATE.G_Methane_Sensors[L_i] >= 20.0 THEN
        IF (GVL_CONFIG.G_Evac_Gas_Zone_Map[L_i] >= 1) AND (GVL_CONFIG.G_Evac_Gas_Zone_Map[L_i] <= GVL_CONFIG.C_MAX_LIGHT_ZONES) THEN
            GVL_STATE.G_Evac_Hazard_Zone[GVL_CONFIG.G_Evac_Gas_Zone_Map[L_i]] := TRUE;
        END_IF;
    END_IF;
END_FOR;

// Публикация агрегированных safety-состояний в единый слой GVL_STATE
GVL_STATE.G_Safety_Leak_Alarm := GVL_ALARM.G_Flood_Alarm_Active;
GVL_STATE.G_Safety_Gas_Alarm := GVL_ALARM.G_Gas_Alarm_Active;
GVL_STATE.G_Safety_Smoke_Alarm := GVL_ALARM.G_Fire_Alarm_Active;

// Integrated water/freeze/valve/operator safety layer
GVL_STATUS.G_Diagnostics.Water_Recovery_Physical_Active := FALSE;
GVL_STATUS.G_Diagnostics.Water_Recovery_Physical_Zone_Name := '';
GVL_STATUS.G_Diagnostics.Water_Localization_Failed := FALSE;
GVL_STATUS.G_Diagnostics.Water_Main_Shutdown_Recommended := FALSE;
GVL_STATUS.G_Diagnostics.Water_Escalation_Text := '';
GVL_STATUS.G_Diagnostics.Water_Close_Fault_Active := FALSE;
GVL_STATUS.G_Diagnostics.Water_Close_Fault_Zone_Name := '';
GVL_STATUS.G_Diagnostics.Water_Close_Fault_Text := '';
GVL_STATUS.G_Diagnostics.Valve_Test_Validation_OK := FALSE;
GVL_STATUS.G_Diagnostics.Valve_Test_Validation_Text := '';
GVL_STATUS.G_Diagnostics.Valve_Test_Forced_Close := FALSE;
GVL_STATUS.G_Diagnostics.Water_Recovery_Target_Zone_Index := 0;
GVL_STATUS.G_Diagnostics.Gas_Recovery_Target_Zone_Index := 0;
GVL_STATUS.G_Diagnostics.Water_Recovery_Selective_Allowed := FALSE;
GVL_STATUS.G_Diagnostics.Gas_Recovery_Selective_Allowed := FALSE;
GVL_STATUS.G_Diagnostics.Water_Recovery_Selective_Text := '';
GVL_STATUS.G_Diagnostics.Gas_Recovery_Selective_Text := '';
GVL_STATUS.G_Diagnostics.Active_Leak_Sensor_Index := 0;
GVL_STATUS.G_Diagnostics.Active_Gas_Sensor_Index := 0;
GVL_STATUS.G_Diagnostics.Active_Leak_Zone_Name := '';
GVL_STATUS.G_Diagnostics.Active_Gas_Zone_Name := '';

FOR L_i := 1 TO GVL_CONSTANTS.C_MAX_FLOOD_SENSORS DO
    IF (GVL_STATUS.G_Diagnostics.Active_Leak_Sensor_Index = 0) AND GVL_STATE.G_Water_Sensors[L_i] THEN
        GVL_STATUS.G_Diagnostics.Active_Leak_Sensor_Index := L_i;
        IF (GVL_CONFIG.G_Evac_Leak_Zone_Map[L_i] >= 1) AND (GVL_CONFIG.G_Evac_Leak_Zone_Map[L_i] <= 32) THEN
            GVL_STATUS.G_Diagnostics.Water_Recovery_Target_Zone_Index := GVL_CONFIG.G_Evac_Leak_Zone_Map[L_i];
            GVL_STATUS.G_Diagnostics.Active_Leak_Zone_Name := GVL_CONFIG.G_Evac_Zone_Names[GVL_CONFIG.G_Evac_Leak_Zone_Map[L_i]];
        END_IF;
        IF GVL_STATUS.G_Diagnostics.Active_Leak_Zone_Name = '' THEN
            GVL_STATUS.G_Diagnostics.Active_Leak_Zone_Name := CONCAT('Leak sensor ', INT_TO_STRING(L_i));
        END_IF;
    END_IF;
END_FOR;
FOR L_i := 1 TO GVL_CONSTANTS.C_MAX_METHANE_SENSORS DO
    IF (GVL_STATUS.G_Diagnostics.Active_Gas_Sensor_Index = 0) AND (GVL_STATE.G_Methane_Sensors[L_i] >= 20.0) THEN
        GVL_STATUS.G_Diagnostics.Active_Gas_Sensor_Index := L_i;
        IF (GVL_CONFIG.G_Evac_Gas_Zone_Map[L_i] >= 1) AND (GVL_CONFIG.G_Evac_Gas_Zone_Map[L_i] <= 32) THEN
            GVL_STATUS.G_Diagnostics.Gas_Recovery_Target_Zone_Index := GVL_CONFIG.G_Evac_Gas_Zone_Map[L_i];
            GVL_STATUS.G_Diagnostics.Active_Gas_Zone_Name := GVL_CONFIG.G_Evac_Zone_Names[GVL_CONFIG.G_Evac_Gas_Zone_Map[L_i]];
        END_IF;
        IF GVL_STATUS.G_Diagnostics.Active_Gas_Zone_Name = '' THEN
            GVL_STATUS.G_Diagnostics.Active_Gas_Zone_Name := CONCAT('Gas sensor ', INT_TO_STRING(L_i));
        END_IF;
    END_IF;
END_FOR;

IF GVL_STATUS.G_Diagnostics.Active_Leak_Sensor_Index > 0 THEN
    GVL_STATUS.G_Diagnostics.Water_Recovery_Selective_Allowed := TRUE;
    GVL_STATUS.G_Diagnostics.Water_Recovery_Selective_Text := CONCAT('Селективное восстановление возможно для зоны ', GVL_STATUS.G_Diagnostics.Active_Leak_Zone_Name);
END_IF;
IF GVL_STATUS.G_Diagnostics.Active_Gas_Sensor_Index > 0 THEN
    GVL_STATUS.G_Diagnostics.Gas_Recovery_Selective_Allowed := TRUE;
    GVL_STATUS.G_Diagnostics.Gas_Recovery_Selective_Text := CONCAT('Газовый контекст локализован в зоне ', GVL_STATUS.G_Diagnostics.Active_Gas_Zone_Name);
END_IF;

FOR L_i := 1 TO 32 DO
    GVL_STATE.G_Water_Zone_Enable[L_i] := FALSE;
    GVL_STATUS.G_Diagnostics.Water_Zone_Open_Fault[L_i] := FALSE;
    GVL_STATUS.G_Diagnostics.Water_Zone_Close_Fault[L_i] := FALSE;
    GVL_STATUS.G_Diagnostics.Water_Zone_Critical_Close_Fault[L_i] := FALSE;
    GVL_STATUS.G_Diagnostics.Water_Zone_Close_Retry_Active[L_i] := FALSE;

    IF NOT GVL_STATE.G_Water_Zone_Enable[L_i] THEN
        IF NOT GVL_STATE.G_Water_Zone_Close_FB[L_i] THEN
            IF GVL_STATUS.G_Diagnostics.Water_Zone_Close_Retry_Count[L_i] < GVL_CONFIG.G_Water_Valve_Close_Retry_Count THEN
                IF (GVL_STATUS.G_System_Time_MS - L_Water_Zone_Close_Last_Retry_MS[L_i]) >= GVL_CONFIG.G_Water_Valve_Close_Retry_Delay_MS THEN
                    GVL_STATUS.G_Diagnostics.Water_Zone_Close_Retry_Active[L_i] := TRUE;
                    GVL_STATUS.G_Diagnostics.Water_Zone_Close_Retry_Count[L_i] := GVL_STATUS.G_Diagnostics.Water_Zone_Close_Retry_Count[L_i] + 1;
                    L_Water_Zone_Close_Last_Retry_MS[L_i] := GVL_STATUS.G_System_Time_MS;
                END_IF;
            ELSE
                GVL_STATUS.G_Diagnostics.Water_Zone_Critical_Close_Fault[L_i] := TRUE;
                GVL_STATUS.G_Diagnostics.Water_Close_Fault_Active := TRUE;
                GVL_STATUS.G_Diagnostics.Water_Close_Fault_Zone_Name := GVL_CONFIG.G_Evac_Zone_Names[L_i];
                IF GVL_STATUS.G_Diagnostics.Water_Close_Fault_Zone_Name = '' THEN
                    GVL_STATUS.G_Diagnostics.Water_Close_Fault_Zone_Name := CONCAT('Water zone ', INT_TO_STRING(L_i));
                END_IF;
                GVL_STATUS.G_Diagnostics.Water_Close_Fault_Text := CONCAT('Не подтверждено аварийное закрытие водяного клапана в зоне ', GVL_STATUS.G_Diagnostics.Water_Close_Fault_Zone_Name);
            END_IF;
        ELSE
            IF GVL_STATUS.G_Diagnostics.Water_Zone_Close_Retry_Count[L_i] > 0 THEN
                GVL_STATUS.G_Diagnostics.Water_Zone_Close_Recovered_After_Retry[L_i] := TRUE;
            END_IF;
            GVL_STATUS.G_Diagnostics.Water_Zone_Close_Retry_Count[L_i] := 0;
        END_IF;
    END_IF;

    IF GVL_CONFIG.G_Water_Valve_Exercise_Enabled AND GVL_STATUS.G_Is_Active_PLC AND
       (GVL_STATUS.G_Current_TOD >= GVL_CONFIG.G_Water_Valve_Exercise_Window_Start) AND
       (GVL_STATUS.G_Current_TOD <= GVL_CONFIG.G_Water_Valve_Exercise_Window_End) AND
       GVL_STATE.G_Water_Zone_Open_FB[L_i] AND
       (GVL_STATE.G_System_Mode = E_System_Operating_Mode.MODE_NORMAL) AND
       (NOT GVL_STATE.G_Safety_Leak_Alarm) AND (NOT GVL_STATE.G_Safety_Gas_Alarm) THEN
        IF (GVL_STATUS.G_System_Time_MS - L_Water_Valve_Last_Exercise_MS[L_i]) >= GVL_CONFIG.G_Water_Valve_Exercise_Interval_MS THEN
            IF L_Water_Valve_Exercise_Until_MS[L_i] = 0 THEN
                L_Water_Valve_Exercise_Until_MS[L_i] := GVL_STATUS.G_System_Time_MS + GVL_CONFIG.G_Water_Valve_Exercise_Duration_MS;
                L_Water_Valve_Last_Exercise_MS[L_i] := GVL_STATUS.G_System_Time_MS;
            END_IF;
        END_IF;
    END_IF;

    IF L_Water_Valve_Exercise_Until_MS[L_i] <> 0 THEN
        IF GVL_STATUS.G_System_Time_MS < L_Water_Valve_Exercise_Until_MS[L_i] THEN
            GVL_STATE.G_Water_Zone_Enable[L_i] := TRUE;
            GVL_STATE.G_Water_Zone_Exercise_Active[L_i] := TRUE;
            GVL_STATUS.G_Diagnostics.Water_Valve_Exercise_Last_Zone := L_i;
            IF GVL_STATE.G_Water_Zone_Open_FB[L_i] THEN
                GVL_STATUS.G_Diagnostics.Water_Valve_Exercise_Last_Result := 'Прокрутка шарового крана подтверждена OPEN_FB';
            ELSE
                GVL_STATUS.G_Diagnostics.Water_Valve_Exercise_Last_Result := 'Прокрутка шарового крана выполняется';
            END_IF;
        ELSE
            L_Water_Valve_Exercise_Until_MS[L_i] := 0;
            GVL_STATE.G_Water_Zone_Enable[L_i] := FALSE;
            GVL_STATE.G_Water_Zone_Exercise_Active[L_i] := FALSE;
            IF GVL_STATE.G_Water_Zone_Close_FB[L_i] THEN
                GVL_STATUS.G_Diagnostics.Water_Valve_Exercise_Last_Result := 'Прокрутка шарового крана завершена и подтверждена CLOSE_FB';
            ELSE
                GVL_STATUS.G_Diagnostics.Water_Valve_Exercise_Last_Result := 'Прокрутка завершена, CLOSE_FB не подтверждён';
            END_IF;
        END_IF;
    END_IF;
END_FOR;

IF GVL_COMMAND.CMD_Water_Selective_Recover THEN
    IF GVL_STATUS.G_Diagnostics.Water_Recovery_Selective_Allowed AND (GVL_STATUS.G_Diagnostics.Water_Recovery_Target_Zone_Index >= 1) AND (GVL_STATUS.G_Diagnostics.Water_Recovery_Target_Zone_Index <= 32) THEN
        GVL_STATE.G_Water_Zone_Enable[GVL_STATUS.G_Diagnostics.Water_Recovery_Target_Zone_Index] := TRUE;
        GVL_STATUS.G_Diagnostics.Water_Recovery_Physical_Active := TRUE;
        GVL_STATUS.G_Diagnostics.Water_Recovery_Physical_Zone_Name := GVL_STATUS.G_Diagnostics.Active_Leak_Zone_Name;
        GVL_STATUS.G_Diagnostics.Water_Valve_Test_Context := CONCAT('Селективный тест воды для зоны ', GVL_STATUS.G_Diagnostics.Active_Leak_Zone_Name);
    ELSE
        GVL_STATUS.G_Diagnostics.Operator_Action_Blocked := TRUE;
        GVL_STATUS.G_Diagnostics.Operator_Block_Reason := 'Селективное восстановление воды недоступно: зона аварии не локализована';
    END_IF;
END_IF;

IF GVL_COMMAND.CMD_Gas_Selective_Recover THEN
    IF GVL_STATUS.G_Diagnostics.Gas_Recovery_Selective_Allowed THEN
        GVL_STATUS.G_Diagnostics.Gas_Valve_Test_Context := CONCAT('Селективный тест газа для зоны ', GVL_STATUS.G_Diagnostics.Active_Gas_Zone_Name);
    ELSE
        GVL_STATUS.G_Diagnostics.Operator_Action_Blocked := TRUE;
        GVL_STATUS.G_Diagnostics.Operator_Block_Reason := 'Селективное восстановление газа недоступно: зона аварии не локализована';
    END_IF;
END_IF;

IF GVL_COMMAND.CMD_Water_Valve_Test_Open THEN
    L_Water_Test_Active := TRUE;
    L_Water_Test_Deadline := GVL_STATUS.G_System_Time_MS + 60000;
    GVL_STATUS.G_Diagnostics.Water_Valve_Test_Mode_Active := TRUE;
    GVL_STATUS.G_Diagnostics.Water_Valve_Test_Deadline_MS := L_Water_Test_Deadline;
END_IF;
IF L_Water_Test_Active THEN
    IF GVL_STATUS.G_System_Time_MS < L_Water_Test_Deadline THEN
        GVL_STATUS.G_Diagnostics.Water_Valve_Test_Remaining_MS := L_Water_Test_Deadline - GVL_STATUS.G_System_Time_MS;
        IF NOT GVL_STATE.G_Safety_Leak_Alarm THEN
            GVL_STATUS.G_Diagnostics.Water_Valve_Test_Validation_OK := TRUE;
            GVL_STATUS.G_Diagnostics.Water_Valve_Test_Validation_Text := CONCAT('Утечка не обнаружена, зона: ', GVL_STATUS.G_Diagnostics.Active_Leak_Zone_Name);
        ELSE
            GVL_STATUS.G_Diagnostics.Water_Valve_Test_Validation_OK := FALSE;
            GVL_STATUS.G_Diagnostics.Water_Valve_Test_Validation_Text := CONCAT('Подтверждение запрещено: активна протечка в зоне ', GVL_STATUS.G_Diagnostics.Active_Leak_Zone_Name);
            GVL_STATUS.G_Diagnostics.Water_Valve_Test_Forced_Close := TRUE;
            GVL_COMMAND.G_Close_Valve_35 := TRUE;
            GVL_COMMAND.G_Close_Valve_36 := TRUE;
            L_Water_Test_Active := FALSE;
            GVL_STATUS.G_Diagnostics.Water_Valve_Test_Mode_Active := FALSE;
        END_IF;
    ELSE
        L_Water_Test_Active := FALSE;
        GVL_STATUS.G_Diagnostics.Water_Valve_Test_Mode_Active := FALSE;
        GVL_COMMAND.G_Close_Valve_35 := TRUE;
        GVL_COMMAND.G_Close_Valve_36 := TRUE;
    END_IF;
END_IF;
IF GVL_COMMAND.CMD_Water_Valve_Test_Close THEN
    L_Water_Test_Active := FALSE;
    GVL_STATUS.G_Diagnostics.Water_Valve_Test_Mode_Active := FALSE;
    GVL_COMMAND.G_Close_Valve_35 := TRUE;
    GVL_COMMAND.G_Close_Valve_36 := TRUE;
END_IF;
IF GVL_COMMAND.CMD_Water_Valve_Test_Confirm AND L_Water_Test_Active THEN
    IF GVL_STATUS.G_Diagnostics.Water_Valve_Test_Validation_OK THEN
        L_Water_Test_Active := FALSE;
        GVL_STATUS.G_Diagnostics.Water_Valve_Test_Mode_Active := FALSE;
    ELSE
        GVL_STATUS.G_Diagnostics.Operator_Action_Blocked := TRUE;
        GVL_STATUS.G_Diagnostics.Operator_Block_Reason := 'Подтверждение водяного теста запрещено: причина аварии не устранена';
    END_IF;
END_IF;

IF GVL_COMMAND.CMD_Gas_Valve_Test_Open THEN
    L_Gas_Test_Active := TRUE;
    L_Gas_Test_Deadline := GVL_STATUS.G_System_Time_MS + 60000;
    GVL_STATUS.G_Diagnostics.Gas_Valve_Test_Mode_Active := TRUE;
    GVL_STATUS.G_Diagnostics.Gas_Valve_Test_Deadline_MS := L_Gas_Test_Deadline;
END_IF;
IF L_Gas_Test_Active THEN
    IF GVL_STATUS.G_System_Time_MS < L_Gas_Test_Deadline THEN
        GVL_STATUS.G_Diagnostics.Gas_Valve_Test_Remaining_MS := L_Gas_Test_Deadline - GVL_STATUS.G_System_Time_MS;
        IF NOT GVL_STATE.G_Safety_Gas_Alarm THEN
            GVL_STATUS.G_Diagnostics.Gas_Valve_Test_Validation_OK := TRUE;
            GVL_STATUS.G_Diagnostics.Gas_Valve_Test_Validation_Text := CONCAT('Газ не обнаружен, зона: ', GVL_STATUS.G_Diagnostics.Active_Gas_Zone_Name);
        ELSE
            GVL_STATUS.G_Diagnostics.Gas_Valve_Test_Validation_OK := FALSE;
            GVL_STATUS.G_Diagnostics.Gas_Valve_Test_Validation_Text := CONCAT('Подтверждение запрещено: активен газ в зоне ', GVL_STATUS.G_Diagnostics.Active_Gas_Zone_Name);
            GVL_STATUS.G_Diagnostics.Gas_Valve_Test_Forced_Close := TRUE;
            GVL_COMMAND.G_Gas_Valve_Close := TRUE;
            L_Gas_Test_Active := FALSE;
            GVL_STATUS.G_Diagnostics.Gas_Valve_Test_Mode_Active := FALSE;
        END_IF;
    ELSE
        L_Gas_Test_Active := FALSE;
        GVL_STATUS.G_Diagnostics.Gas_Valve_Test_Mode_Active := FALSE;
        GVL_COMMAND.G_Gas_Valve_Close := TRUE;
    END_IF;
END_IF;
IF GVL_COMMAND.CMD_Gas_Valve_Test_Close THEN
    L_Gas_Test_Active := FALSE;
    GVL_STATUS.G_Diagnostics.Gas_Valve_Test_Mode_Active := FALSE;
    GVL_COMMAND.G_Gas_Valve_Close := TRUE;
END_IF;
IF GVL_COMMAND.CMD_Gas_Valve_Test_Confirm AND L_Gas_Test_Active THEN
    IF GVL_STATUS.G_Diagnostics.Gas_Valve_Test_Validation_OK THEN
        L_Gas_Test_Active := FALSE;
        GVL_STATUS.G_Diagnostics.Gas_Valve_Test_Mode_Active := FALSE;
    ELSE
        GVL_STATUS.G_Diagnostics.Operator_Action_Blocked := TRUE;
        GVL_STATUS.G_Diagnostics.Operator_Block_Reason := 'Подтверждение газового теста запрещено: причина аварии не устранена';
    END_IF;
END_IF;

IF GVL_STATE.G_Safety_Leak_Alarm THEN
    FOR L_i := 1 TO 32 DO
        IF GVL_STATUS.G_Diagnostics.Water_Zone_Critical_Close_Fault[L_i] THEN
            GVL_STATUS.G_Diagnostics.Water_Localization_Failed := TRUE;
            GVL_STATUS.G_Diagnostics.Water_Main_Shutdown_Recommended := TRUE;
            IF GVL_CONFIG.G_Evac_Zone_Names[L_i] <> '' THEN
                GVL_STATUS.G_Diagnostics.Water_Escalation_Text := CONCAT('Реальная протечка не локализована, рекомендуется перекрыть общий ввод воды: ', GVL_CONFIG.G_Evac_Zone_Names[L_i]);
            ELSE
                GVL_STATUS.G_Diagnostics.Water_Escalation_Text := CONCAT('Реальная протечка не локализована, рекомендуется перекрыть общий ввод воды: зона ', INT_TO_STRING(L_i));
            END_IF;
        END_IF;
    END_FOR;
END_IF;
IF GVL_STATUS.G_Diagnostics.Water_Main_Shutdown_Recommended THEN
    GVL_STATUS.G_Diagnostics.Operator_Action_Blocked := TRUE;
    GVL_STATUS.G_Diagnostics.Operator_Block_Reason := GVL_STATUS.G_Diagnostics.Water_Escalation_Text;
END_IF;

IF GVL_STATE.G_Freeze_Hardware_Degraded THEN
    GVL_STATUS.G_Diagnostics.Freeze_Hardware_Event_Pending := TRUE;
END_IF;
// >>> BULK_SYNC_ANCHOR: PRG_Safety <<<
          
END_PROGRAM

PROGRAM PRG_Security
  VAR
    L_i : INT;
    L_Motion_Sensors_16 : ARRAY[1..16] OF BOOL;
    fbSecurityManager : FB_Security_System_Manager;
    fbAccessControl : FB_Access_Control;
  END_VAR

            FOR L_i := 1 TO 16 DO
    L_Motion_Sensors_16[L_i] := L_Motion_Sensors_16[L_i];
END_FOR;
// 7. Система безопасности (Охранная сигнализация)
fbSecurityManager(
    VI_System_Time_MS := GVL_STATUS.G_System_Time_MS,
    VI_IsActivePLC := GVL_STATUS.G_Is_Active_PLC,
    VI_Motion_Sensors := L_Motion_Sensors_16,
    VI_Door_Sensors := GVL_STATE.G_Door_Sensors,
    VI_Window_Sensors := GVL_STATE.G_Window_Sensors,
    VI_Arm_Request := GVL_COMMAND.G_Arm_Req,
    VI_Disarm_Request := GVL_COMMAND.G_Disarm_Req,
    VI_PIN_Code := GVL_COMMAND.G_PIN_Code,
    VI_RFID_Tag := GVL_COMMAND.G_RFID_Tag,
    VI_2FA_Code := GVL_COMMAND.G_2FA_Code_In,
    VI_Config := GVL_CONFIG.G_Security_Config,
    VI_Bypass_Motion := GVL_CONFIG.G_Security_Config.bypass_motion,
    VI_Bypass_Doors := GVL_CONFIG.G_Security_Config.bypass_doors,
    VI_Bypass_Windows := GVL_CONFIG.G_Security_Config.bypass_windows,
    VI_Current_TOD := GVL_STATUS.G_Current_TOD,
    VO_Armed => GVL_ALARM.G_Security_Armed,
    VO_Alarm_Active => GVL_ALARM.G_Security_Alarm,
    VO_Siren_Active => GVL_ALARM.G_Security_Siren,
    VO_Status_Msg => GVL_STATUS.G_Security_Status_Msg,
    VO_Send_Code_Req => GVL_COMMAND.G_Send_2FA_Req,
    VO_Code_To_Send => GVL_COMMAND.G_2FA_Code_Out
);

// 7.1 Контроль доступа (СКУД)
fbAccessControl(
    VI_System_Time_MS := GVL_STATUS.G_System_Time_MS,
    VI_IsActivePLC := GVL_STATUS.G_Is_Active_PLC,
    VI_Armed := GVL_ALARM.G_Security_Armed,
    VI_Gate_Open_Req := GVL_CONFIG.G_HMI_Gate_Open_Req,
    VI_Wicket_Open_Req := GVL_CONFIG.G_HMI_Wicket_Open_Req,
    VI_Lock_1_Open_Req := GVL_CONFIG.G_HMI_Lock_1_Open_Req,
    VI_Lock_1_Close_Req := GVL_CONFIG.G_HMI_Lock_1_Close_Req,
    VI_Lock_2_Open_Req := GVL_CONFIG.G_HMI_Lock_2_Open_Req,
    VI_Lock_2_Close_Req := GVL_CONFIG.G_HMI_Lock_2_Close_Req,
    VI_PIN_Code := GVL_COMMAND.G_PIN_Code,
    VI_RFID_Tag := GVL_COMMAND.G_RFID_Tag,
    VI_Access_Codes := GVL_Retain.G_Access_Codes,
    VI_RFID_Tags := GVL_Retain.G_RFID_Tags,
    VI_Config := GVL_CONFIG.G_Security_Config,
    VO_Gate_Open => GVL_COMMAND.G_Gate_Open,
    VO_Wicket_Open => GVL_COMMAND.G_Wicket_Open,
    VO_Lock_1_Open => GVL_COMMAND.G_Lock_1_Open,
    VO_Lock_1_Close => GVL_COMMAND.G_Lock_1_Close,
    VO_Lock_2_Open => GVL_COMMAND.G_Lock_2_Open,
    VO_Lock_2_Close => GVL_COMMAND.G_Lock_2_Close
);
// >>> BULK_SYNC_ANCHOR: PRG_Security <<<
          
END_PROGRAM

